# B&R Automation Studio project NAINV104C00R8L515F00 (part 17)

#### InputRef_Link.var - Change By Project
```iecst
(*2020-09-22*)
(**)
(*User Folder*)
VAR
	p_eUsrFolderStat : REFERENCE TO eUsrFolderAction;
	p_eUsrFolderStatus : REFERENCE TO eFBStatus;
END_VAR
(**)
(*Hardware Info*)
VAR
	p_eHWInfoStat : REFERENCE TO eHWInfoAction;
	p_eHWInfoStatus : REFERENCE TO eFBStatus;
	p_sHWInfoIPAddr : REFERENCE TO STRING[15];
	p_sHWInfoSubnetMask : REFERENCE TO STRING[15];
	p_udiHWInfoEthMode : REFERENCE TO UDINT;
END_VAR
(**)
(*Library Version*)
VAR
	p_eLibVerStat : REFERENCE TO eLibVerAction;
	p_eLibVerStatus : REFERENCE TO eFBStatus;
END_VAR
(**)
(*Nutek Parameter*)
VAR
	p_eNtParamStat : REFERENCE TO eNtParamAction;
	p_eNtParamStatus : REFERENCE TO eFBStatus;
END_VAR
(**)
(*Machine Parameter*)
VAR
	p_eMcParamStat : REFERENCE TO eMcParamAction;
	p_eMcParamStatus : REFERENCE TO eFBStatus;
END_VAR
(**)
(*Product Recipe*)
VAR
	p_eProdRcpStat : REFERENCE TO eProdRcpAction;
	p_eProdRcpStatus : REFERENCE TO eFBStatus;
END_VAR
(**)
(*Mp Product Recipe*)
VAR
	p_eMpProdRcpStat : REFERENCE TO eMpProdRcpAction;
	p_eMpProdRcpStatus : REFERENCE TO eFBStatus;
END_VAR
(**)
(*User Management*)
VAR
	p_eUsrMgmtStat : REFERENCE TO eUsrMgmtAction;
	p_eUsrMgmtStatus : REFERENCE TO eFBStatus;
END_VAR
(**)
(*Alarm Log*)
VAR
	p_eAlarmStat : REFERENCE TO eAlarmAction;
	p_eAlarmStatus : REFERENCE TO eFBStatus;
END_VAR
(**)
(*Hermes*)
VAR
	p_eHermesStat : REFERENCE TO eHermesAction;
	p_eHermesStatus : REFERENCE TO eFBStatus;
END_VAR
(**)
VAR
	p_eRmtHermesStat : REFERENCE TO eHermesAction;
	p_eRmtHermesStatus : REFERENCE TO eFBStatus;
END_VAR
(**)
VAR
	p_eUSHermesStat : REFERENCE TO eHermesAction;
	p_eUSHermesStatus : REFERENCE TO eFBStatus;
END_VAR
(**)
VAR
	p_eDSHermesStat : REFERENCE TO eHermesAction;
	p_eDSHermesStatus : REFERENCE TO eFBStatus;
END_VAR
(**)
(*Auto Width*)
VAR
	p_eAWStat : REFERENCE TO eAWAction;
	p_eAWStatus : REFERENCE TO eFBStatus;
END_VAR
(**)
(*User Interface*)
VAR
	p_eUIStat : REFERENCE TO eUIAction;
	p_eUIStatus : REFERENCE TO eFBStatus;
END_VAR
```

#### Act_Link.st - Change By Project
```iecst
(** 2018-12-12 **)
ACTION Act_Link:

END_ACTION
```

#### Cyclic.st - Do Not Change!!!
```iecst
(** 2019-03-29 **)
PROGRAM _CYCLIC

	IF bInitDone = FALSE THEN
		bInitDone	:= TRUE;

		Act_InitLocal;
		Act_InitGlobal;

	ELSIF bInitialDone = FALSE THEN
		bInitialDone	:= TRUE;

		Act_Initial;

	ELSE

		Act_LinkAction;
		Act_Action;
		Act_Link;
		Act_Main;

	END_IF

END_PROGRAM
```

#### Act_InitLocal.st - Do Not Change!!!
```iecst
(** 2020-09-22 **)
ACTION Act_InitLocal:

	//Input Reference Link To Local Variable
	p_eAct ACCESS ADR(eAct);
	p_tyNtParamCurr ACCESS ADR(tyNtParamCurr);
	p_tyMcParamCurr ACCESS ADR(tyMcParamCurr);

	p_bUIMismatchOverWriteConfig ACCESS ADR(bMismatchOverWriteConfig);
	p_bUITempAddrFillDone ACCESS ADR(bTempAddrFillDone);
	p_bUIChgConfigDone ACCESS ADR(bChgConfigDone);
	p_bUIOverwriteIP ACCESS ADR(bOverwriteIP);
	p_bUIOverwriteSubnet ACCESS ADR(bOverwriteSubnet);
	p_bUIOverwriteEthMode ACCESS ADR(bOverwriteEthMode);

END_ACTION
```

#### Act_Initial.st - Do Not Change!!!
```iecst
(** 2019-02-20 **)
ACTION Act_Initial:

	//Initial
	sStatTxt	:= a_sStatText[eStat];

END_ACTION
```

#### Act_Action.st - Do Not Change!!!
```iecst
(** 2019-03-25 **)
ACTION Act_Action:

	//Reset Done
	IF eStatus = Done AND p_eAct = StartupActIdle THEN
		eStat	:= StartupActIdle;
	END_IF

	//Set p_eAct
	IF eStatus = Idle THEN
		eStat	:= p_eAct;
	END_IF

END_ACTION
```

#### Act_Main.st - Change By Project
```iecst
(** 2019-03-28 **)
ACTION Act_Main:

	//Main
	CASE eStat OF

		StartupActIdle:
			IF eStatus <> Idle THEN	//Reset Data
				//Private
				eStartupStep1	:= StartupStepUsrFolder;
				bRun			:= FALSE;
				usiStep			:= 0;

				sStatTxt	:= a_sStatText[eStat];

			END_IF

			eStatus	:= Idle;

		StartupActRun:
			IF eStatus = Idle OR eStatus = Busy THEN

				eStatus	:= Busy;

				sStatTxt	:= a_sStatText[eStat];

				bRun	:= TRUE;

				CASE eStartupStep1 OF

					StartupStepUsrFolder:
						Act_Main_UsrFolder;

					StartupStepParameter:
						Act_Main_Parameter;

					StartupStepGetHWInfo:
						Act_Main_GetHWInfo;

					StartupStepLibVer:
						Act_Main_LibVer;

					StartupStepRecipe:
						Act_Main_Recipe;

					StartupStepUsrMgmt:
						Act_Main_UsrMgmt;

					StartupStepBffr:
						Act_Main_Bffr;

					StartupStepAlarm:
						Act_Main_Alarm;

					StartupStepHermes:
						Act_Main_Hermes;

					StartupStepSDOWrite:
						Act_Main_SDOWrite;

					StartupStepSetupUI:
						Act_Main_SetupUI;

					StartupStepDone:
						Act_Main_Done;

				END_CASE

				sStepTxt	:= a_sStepText[eStartupStep1];

			END_IF

	END_CASE

END_ACTION
```

#### Package Logical/Startup/Startup/Act_Main - Change By Project

#### Act_Main_UsrFolder.st
```iecst
(** 2019-05-09 **)
ACTION Act_Main_UsrFolder:

	CASE usiStep OF
		0:
			eUsrFolderAct	:= UsrFolderActCreateUsrDir;

			IF (p_eUsrFolderStatus = Done) AND (p_eUsrFolderStat = UsrFolderActCreateUsrDir) THEN

				eUsrFolderAct	:= UsrFolderActIdle;
				usiStep			:= 1;

			ELSIF p_eUsrFolderStatus = Error THEN

				eUsrFolderAct	:= UsrFolderActIdle;
				eStartupStep1	:= StartupStepParameter;

			END_IF

		1:
			eUsrFolderAct	:= UsrFolderActCreatePrivateDir;

			IF (p_eUsrFolderStatus = Done) AND (p_eUsrFolderStat = UsrFolderActCreatePrivateDir) THEN

				eUsrFolderAct	:= UsrFolderActIdle;
				usiStep			:= 2;

			ELSIF p_eUsrFolderStatus = Error THEN

				eUsrFolderAct	:= UsrFolderActIdle;
				usiStep			:= 0;
				eStartupStep1	:= StartupStepParameter;

			END_IF

		2:
			eUsrFolderAct	:= UsrFolderActCreateLogDir;

			IF (p_eUsrFolderStatus = Done) AND (p_eUsrFolderStat = UsrFolderActCreateLogDir) THEN

				eUsrFolderAct	:= UsrFolderActIdle;
				usiStep			:= 3;

			ELSIF p_eUsrFolderStatus = Error THEN

				eUsrFolderAct	:= UsrFolderActIdle;
				usiStep			:= 0;
				eStartupStep1	:= StartupStepParameter;

			END_IF

		3:
			eUsrFolderAct	:= UsrFolderActCreateLCSDir;

			IF (p_eUsrFolderStatus = Done) AND (p_eUsrFolderStat = UsrFolderActCreateLCSDir) THEN

				eUsrFolderAct	:= UsrFolderActIdle;
				usiStep			:= 0;
				eStartupStep1	:= StartupStepParameter;

			ELSIF p_eUsrFolderStatus = Error THEN

				eUsrFolderAct	:= UsrFolderActIdle;
				usiStep			:= 0;
				eStartupStep1	:= StartupStepParameter;

			END_IF

	END_CASE

END_ACTION
```

#### Act_Main_GetHWInfo.st
```iecst
(** 2020-10-05 **)
ACTION Act_Main_GetHWInfo:

	CASE usiStep OF
		0:
			eHWInfoAct	:= HWInfoActGetIPAddr;

			IF (p_eHWInfoStatus = Done) AND (p_eHWInfoStat = HWInfoActGetIPAddr) THEN

				eHWInfoAct		:= HWInfoActIdle;
				usiStep			:= 1;

			ELSIF p_eHWInfoStatus = Error THEN

				eHWInfoAct		:= HWInfoActIdle;
				eStartupStep1	:= StartupStepLibVer;

			END_IF

		1:
			eHWInfoAct	:= HWInfoActGetMacAddr;

			IF (p_eHWInfoStatus = Done) AND (p_eHWInfoStat = HWInfoActGetMacAddr) THEN

				eHWInfoAct		:= HWInfoActIdle;
				usiStep			:= 2;

			ELSIF p_eHWInfoStatus = Error THEN

				eHWInfoAct		:= HWInfoActIdle;
				usiStep			:= 0;
				eStartupStep1	:= StartupStepLibVer;

			END_IF

		2:
			eHWInfoAct	:= HWInfoActGetSubnetMask;

			IF (p_eHWInfoStatus = Done) AND (p_eHWInfoStat = HWInfoActGetSubnetMask) THEN

				eHWInfoAct		:= HWInfoActIdle;

				IF DiagCpuIsSimulated() = TRUE THEN
					usiStep			:= 0;
					eStartupStep1	:= StartupStepLibVer;
				ELSE
					usiStep			:= 3;
				END_IF

			ELSIF p_eHWInfoStatus = Error THEN

				eHWInfoAct		:= HWInfoActIdle;
				usiStep			:= 0;
				eStartupStep1	:= StartupStepLibVer;

			END_IF

		3:
			eHWInfoAct	:= HWInfoActGetEthConfigMode;

			IF (p_eHWInfoStatus = Done) AND (p_eHWInfoStat = HWInfoActGetEthConfigMode) THEN

				eHWInfoAct		:= HWInfoActIdle;

				bGetConfigDone	:= TRUE;

				IF (p_tyMcParamCurr.eNetworkMod = UDINT_TO_DINT(p_udiHWInfoEthMode))  THEN
					IF p_udiHWInfoEthMode = DINT_TO_UDINT(IPFromDHCPServer) THEN
						usiStep			:= 0;
						eStartupStep1	:= StartupStepLibVer;
					ELSE
						IF (p_tyMcParamCurr.sIPAddr <> p_sHWInfoIPAddr) OR (p_tyMcParamCurr.sSubnetMask <> p_sHWInfoSubnetMask) THEN
							IF p_bUITempAddrFillDone AND p_bUIMismatchOverWriteConfig THEN
								IF (p_tyMcParamCurr.sIPAddr <> p_sHWInfoIPAddr) THEN
									usiStep			:= 5;  //mismatch ip
								ELSE
									usiStep			:= 6;  //mismatch subnet
								END_IF
							END_IF
						ELSE
							usiStep			:= 0;
							eStartupStep1	:= StartupStepLibVer;
						END_IF
					END_IF

				ELSE
					IF p_bUITempAddrFillDone AND p_bUIMismatchOverWriteConfig THEN
						usiStep			:= 4;
					END_IF
				END_IF

			ELSIF p_eHWInfoStatus = Error THEN

				eHWInfoAct		:= HWInfoActIdle;
				usiStep			:= 0;
				eStartupStep1	:= StartupStepLibVer;

			END_IF

		4:
			eHWInfoAct	:= HWInfoActSetEthConfigMode;

			IF (p_eHWInfoStatus = Done) AND (p_eHWInfoStat = HWInfoActSetEthConfigMode) THEN

				eHWInfoAct		:= HWInfoActIdle;

				IF (p_tyMcParamCurr.eNetworkMod = IPFromDHCPServer) THEN
					usiStep			:= 7;
					bMismatchSetConfigDone	:= TRUE;
				ELSE
					usiStep			:= 5;
				END_IF

			ELSIF p_eHWInfoStatus = Error THEN

				eHWInfoAct		:= HWInfoActIdle;
				usiStep			:= 0;
				eStartupStep1	:= StartupStepLibVer;

			END_IF

		5:
			eHWInfoAct	:= HWInfoActSetIPAddr;

			IF (p_eHWInfoStatus = Done) AND (p_eHWInfoStat = HWInfoActSetIPAddr) THEN

				eHWInfoAct		:= HWInfoActIdle;

				IF (p_tyMcParamCurr.sSubnetMask <> p_sHWInfoSubnetMask) THEN
					usiStep			:= 6;
				ELSE
					usiStep			:= 7;
					bMismatchSetConfigDone	:= TRUE;
				END_IF

			ELSIF p_eHWInfoStatus = Error THEN

				eHWInfoAct		:= HWInfoActIdle;
				usiStep			:= 0;
				eStartupStep1	:= StartupStepLibVer;

			END_IF

		6:
			eHWInfoAct	:= HWInfoActSetSubnetMask;

			IF (p_eHWInfoStatus = Done) AND (p_eHWInfoStat = HWInfoActSetSubnetMask) THEN

				eHWInfoAct		:= HWInfoActIdle;
				usiStep			:= 7;

				bMismatchSetConfigDone	:= TRUE;

			ELSIF p_eHWInfoStatus = Error THEN

				eHWInfoAct		:= HWInfoActIdle;
				usiStep			:= 0;
				eStartupStep1	:= StartupStepLibVer;

			END_IF

		7:
			IF p_bUIChgConfigDone THEN
				IF p_bUIOverwriteEthMode THEN
					usiStep			:= 8; //Overwrite Network Mode
				ELSIF p_bUIOverwriteIP THEN
					usiStep			:= 9; //Overwrite IP
				ELSIF p_bUIOverwriteSubnet THEN
					usiStep			:= 10; //Overwrite Subnet
				ELSE
					usiStep			:= 12; //Load Machine Setting
				END_IF
			END_IF

		8:
			eHWInfoAct	:= HWInfoActSetEthConfigMode;

			IF (p_eHWInfoStatus = Done) AND (p_eHWInfoStat = HWInfoActSetEthConfigMode) THEN

				eHWInfoAct		:= HWInfoActIdle;

				IF p_bUIOverwriteIP THEN
					usiStep			:= 9;
				ELSIF p_bUIOverwriteSubnet THEN
					usiStep			:= 10;
				ELSE
					usiStep			:= 11;
				END_IF

			ELSIF p_eHWInfoStatus = Error THEN

				eHWInfoAct		:= HWInfoActIdle;
				usiStep			:= 0;
				eStartupStep1	:= StartupStepLibVer;

			END_IF

		9:
			eHWInfoAct	:= HWInfoActSetIPAddr;

			IF (p_eHWInfoStatus = Done) AND (p_eHWInfoStat = HWInfoActSetIPAddr) THEN

				eHWInfoAct		:= HWInfoActIdle;

				IF p_bUIOverwriteSubnet THEN
					usiStep			:= 10;
				ELSE
					usiStep			:= 11;
				END_IF

			ELSIF p_eHWInfoStatus = Error THEN

				eHWInfoAct		:= HWInfoActIdle;
				usiStep			:= 0;
				eStartupStep1	:= StartupStepLibVer;

			END_IF

		10:
			eHWInfoAct	:= HWInfoActSetSubnetMask;

			IF (p_eHWInfoStatus = Done) AND (p_eHWInfoStat = HWInfoActSetSubnetMask) THEN

				eHWInfoAct		:= HWInfoActIdle;
				usiStep			:= 11;

			ELSIF p_eHWInfoStatus = Error THEN

				eHWInfoAct		:= HWInfoActIdle;
				usiStep			:= 0;
				eStartupStep1	:= StartupStepLibVer;

			END_IF

		11:

			eMcParamAct	:= McParamActWrite;

			IF (p_eMcParamStatus = Done) AND (p_eMcParamStat = McParamActWrite) THEN

				eMcParamAct		:= McParamActIdle;

				usiStep			:= 12;

			ELSIF p_eMcParamStatus = Error THEN

				eMcParamAct		:= McParamActIdle;
				usiStep			:= 0;
				eStartupStep1	:= StartupStepLibVer;

			END_IF

		12:
			eHWInfoAct	:= HWInfoActGetIPAddr;

			IF (p_eHWInfoStatus = Done) AND (p_eHWInfoStat = HWInfoActGetIPAddr) THEN

				eHWInfoAct		:= HWInfoActIdle;
				usiStep			:= 13;

			ELSIF p_eHWInfoStatus = Error THEN

				eHWInfoAct		:= HWInfoActIdle;
				usiStep			:= 0;
				eStartupStep1	:= StartupStepLibVer;

			END_IF

		13:
			eHWInfoAct	:= HWInfoActGetSubnetMask;

			IF (p_eHWInfoStatus = Done) AND (p_eHWInfoStat = HWInfoActGetSubnetMask) THEN

				eHWInfoAct		:= HWInfoActIdle;
				usiStep			:= 0;
				eStartupStep1	:= StartupStepLibVer;

			ELSIF p_eHWInfoStatus = Error THEN

				eHWInfoAct		:= HWInfoActIdle;
				usiStep			:= 0;
				eStartupStep1	:= StartupStepLibVer;

			END_IF

	END_CASE

END_ACTION
```

#### Act_Main_LibVer.st
```iecst
(** 2019-03-28 **)
ACTION Act_Main_LibVer:

	CASE usiStep OF
		0:
			eLibVerAct	:= LibVerActCreateDir;

			IF (p_eLibVerStatus = Done) AND (p_eLibVerStat = LibVerActCreateDir) THEN

				eLibVerAct		:= LibVerActIdle;
				usiStep			:= 1;

			ELSIF p_eLibVerStatus = Error THEN

				eLibVerAct		:= LibVerActIdle;
				eStartupStep1	:= StartupStepRecipe;

			END_IF

		1:
			eLibVerAct	:= LibVerActReadChk;

			IF (p_eLibVerStatus = Done) AND (p_eLibVerStat = LibVerActReadChk) THEN

				eLibVerAct		:= LibVerActIdle;
				usiStep			:= 0;
				eStartupStep1	:= StartupStepRecipe;

			ELSIF p_eLibVerStatus = Error THEN

				eLibVerAct		:= LibVerActIdle;
				usiStep			:= 0;
				eStartupStep1	:= StartupStepRecipe;

			END_IF

	END_CASE

END_ACTION
```

#### Act_Main_Parameter.st
```iecst
(** 2019-03-28 **)
ACTION Act_Main_Parameter:

	CASE usiStep OF
		0:
			eNtParamAct	:= NtParamActCreateDir;

			IF (p_eNtParamStatus = Done) AND (p_eNtParamStat = NtParamActCreateDir) THEN

				eNtParamAct			:= NtParamActIdle;
				usiStep				:= 1;

			ELSIF p_eNtParamStatus = Error THEN

				bNtSettingsLoadDone	:= TRUE;
				eNtParamAct			:= NtParamActIdle;
				usiStep				:= 2;

			END_IF

		1:
			eNtParamAct	:= NtParamActRead;

			IF (p_eNtParamStatus = Done) AND (p_eNtParamStat = NtParamActRead) THEN

				bNtSettingsLoadDone	:= TRUE;
				eNtParamAct			:= NtParamActIdle;
				usiStep				:= 2;

			ELSIF p_eNtParamStatus = Error THEN

				bNtSettingsLoadDone	:= TRUE;
				eNtParamAct			:= NtParamActIdle;
				usiStep				:= 2;

			END_IF

		2:
			eMcParamAct	:= McParamActCreateDir;

			IF (p_eMcParamStatus = Done) AND (p_eMcParamStat = McParamActCreateDir) THEN

				eMcParamAct		:= McParamActIdle;
				usiStep			:= 3;

			ELSIF p_eMcParamStatus = Error THEN

				eMcParamAct		:= McParamActIdle;
				usiStep			:= 0;
				eStartupStep1	:= StartupStepGetHWInfo;

			END_IF

		3:
			eMcParamAct	:= McParamActRead;

			IF (p_eMcParamStatus = Done) AND (p_eMcParamStat = McParamActRead) THEN

				eMcParamAct		:= McParamActIdle;
				usiStep			:= 0;
				eStartupStep1	:= StartupStepGetHWInfo;

			ELSIF p_eMcParamStatus = Error THEN

				eMcParamAct		:= McParamActIdle;
				usiStep			:= 0;
				eStartupStep1	:= StartupStepGetHWInfo;

			END_IF

	END_CASE

END_ACTION
```

#### Act_Main_Recipe.st
```iecst
(** 2019-05-04 **)
ACTION Act_Main_Recipe:

	CASE usiStep OF
		0:
			eProdRcpAct	:= ProdRcpActCreateDir;

			IF (p_eProdRcpStatus = Done) AND (p_eProdRcpStat = ProdRcpActCreateDir) THEN

				eProdRcpAct		:= ProdRcpActIdle;
				usiStep			:= 1;

			ELSIF p_eProdRcpStatus = Error THEN

				eProdRcpAct		:= ProdRcpActIdle;
				usiStep			:= 10;

			END_IF

		1:
			eProdRcpAct	:= ProdRcpActGetList;

			IF (p_eProdRcpStatus = Done) AND (p_eProdRcpStat = ProdRcpActGetList) THEN

				eProdRcpAct		:= ProdRcpActIdle;
				usiStep			:= 2;

			ELSIF p_eProdRcpStatus = Error THEN

				eProdRcpAct		:= ProdRcpActIdle;
				usiStep			:= 10;

			END_IF

		2:
			eProdRcpAct	:= ProdRcpActReadCurrRcp;

			IF (p_eProdRcpStatus = Done) AND (p_eProdRcpStat = ProdRcpActReadCurrRcp) THEN

				eProdRcpAct		:= ProdRcpActIdle;
				usiStep			:= 10;

			ELSIF p_eProdRcpStatus = Error THEN

				eProdRcpAct		:= ProdRcpActIdle;
				usiStep			:= 10;

			END_IF

		10:
			eMpProdRcpAct	:= MpProdRcpActCreateDir;

			IF (p_eMpProdRcpStatus = Done) AND (p_eMpProdRcpStat = MpProdRcpActCreateDir) THEN

				eMpProdRcpAct	:= MpProdRcpActIdle;
				usiStep			:= 0;
				eStartupStep1	:= StartupStepUsrMgmt;

			ELSIF p_eProdRcpStatus = Error THEN

				eMpProdRcpAct	:= MpProdRcpActIdle;
				usiStep			:= 0;
				eStartupStep1	:= StartupStepUsrMgmt;

			END_IF

	END_CASE

END_ACTION
```

#### Act_Main_UsrMgmt.st
```iecst
(** 2019-03-28 **)
ACTION Act_Main_UsrMgmt:

	CASE usiStep OF
		0:
			eUsrMgmtAct	:= UsrMgmtActCreateDir;

			IF (p_eUsrMgmtStatus = Done) AND (p_eUsrMgmtStat = UsrMgmtActCreateDir) THEN

				eUsrMgmtAct		:= UsrMgmtActIdle;
				usiStep			:= 1;

			ELSIF p_eUsrMgmtStatus = Error THEN

				eUsrMgmtAct		:= UsrMgmtActIdle;
				eStartupStep1	:= StartupStepBffr;

			END_IF

		1:
			eUsrMgmtAct	:= UsrMgmtActReadData;

			IF (p_eUsrMgmtStatus = Done) AND (p_eUsrMgmtStat = UsrMgmtActReadData) THEN

				eUsrMgmtAct		:= UsrMgmtActIdle;
				usiStep			:= 2;

			ELSIF p_eUsrMgmtStatus = Error THEN

				eUsrMgmtAct		:= UsrMgmtActIdle;
				usiStep			:= 0;
				eStartupStep1	:= StartupStepBffr;

			END_IF

		2:
			eUsrMgmtAct	:= UsrMgmtActLogout;

			IF (p_eUsrMgmtStatus = Done) AND (p_eUsrMgmtStat = UsrMgmtActLogout) THEN

				eUsrMgmtAct		:= UsrMgmtActIdle;
				usiStep			:= 0;
				eStartupStep1	:= StartupStepBffr;

			ELSIF p_eUsrMgmtStatus = Error THEN

				eUsrMgmtAct		:= UsrMgmtActIdle;
				usiStep			:= 0;
				eStartupStep1	:= StartupStepBffr;

			END_IF

	END_CASE

END_ACTION
```

#### Act_Main_Bffr.st
```iecst
(** 2013-04-26 **)
ACTION Act_Main_Bffr:

	eStartupStep1	:= StartupStepAlarm;

END_ACTION
```

#### Act_Main_Alarm.st
```iecst
(** 2019-03-28 **)
ACTION Act_Main_Alarm:

	CASE usiStep OF
		0:
			eAlarmAct	:= AlarmActCreateDir;

			IF (p_eAlarmStatus = Done) AND (p_eAlarmStat = AlarmActCreateDir) THEN

				eAlarmAct		:= AlarmActIdle;
				usiStep			:= 1;

			ELSIF p_eAlarmStatus = Error THEN

				eAlarmAct		:= AlarmActIdle;
				usiStep			:= 0;
				eStartupStep1	:= StartupStepHermes;

			END_IF

		1:
			eAlarmAct	:= AlarmActDeleteOldLog;

			IF (p_eAlarmStatus = Done) AND (p_eAlarmStat = AlarmActDeleteOldLog) THEN

				eAlarmAct		:= AlarmActIdle;
				usiStep			:= 2;

			ELSIF p_eAlarmStatus = Error THEN

				eAlarmAct		:= AlarmActIdle;
				usiStep			:= 0;
				eStartupStep1	:= StartupStepHermes;

			END_IF

		2:
			eAlarmAct	:= AlarmActReadHistory;

			IF (p_eAlarmStatus = Done) AND (p_eAlarmStat = AlarmActReadHistory) THEN

				eAlarmAct		:= AlarmActIdle;
				usiStep			:= 3;

			ELSIF p_eAlarmStatus = Error THEN

				eAlarmAct		:= AlarmActIdle;
				usiStep			:= 0;
				eStartupStep1	:= StartupStepHermes;

			END_IF

		3:
			eAlarmAct	:= AlarmActBGStartLog;

			IF (p_eAlarmStatus = Done) AND (p_eAlarmStat = AlarmActBGStartLog) THEN

				eAlarmAct		:= AlarmActIdle;
				usiStep			:= 0;
				eStartupStep1	:= StartupStepHermes;

			ELSIF p_eAlarmStatus = Error THEN

				eAlarmAct		:= AlarmActIdle;
				usiStep			:= 0;
				eStartupStep1	:= StartupStepHermes;

			END_IF

	END_CASE

END_ACTION
```

#### Act_Main_Hermes.st
```iecst
(** 2019-05-04 **)
ACTION Act_Main_Hermes:

	CASE usiStep OF
		0:
			eHermesAct	:= HermesActCreateDir;

			IF (p_eHermesStatus = Done) AND (p_eHermesStat = HermesActCreateDir) THEN

				eHermesAct		:= HermesActIdle;
				usiStep			:= 1;

			ELSIF p_eHermesStatus = Error THEN

				eHermesAct		:= HermesActIdle;
				usiStep			:= 10;

			END_IF

		1:
			eHermesAct	:= HermesActReadRetainLane1; //HermesActReadRetain;

			IF (p_eHermesStatus = Done) AND (p_eHermesStat = HermesActReadRetainLane1) THEN

				eHermesAct		:= HermesActIdle;
				usiStep			:= 2;

			ELSIF p_eHermesStatus = Error THEN

				eHermesAct		:= HermesActIdle;
				usiStep			:= 10;

			END_IF

		2:
			eHermesAct	:= HermesActReadConfig;

			IF (p_eHermesStatus = Done) AND (p_eHermesStat = HermesActReadConfig) THEN

				eHermesAct		:= HermesActIdle;
				usiStep			:= 10;

			ELSIF p_eHermesStatus = Error THEN

				eHermesAct		:= HermesActIdle;
				usiStep			:= 10;

			END_IF

		10:
			eRmtHermesAct	:= HermesActDeleteOldLog;

			IF (p_eRmtHermesStatus = Done) AND (p_eRmtHermesStat = HermesActDeleteOldLog) THEN

				eRmtHermesAct	:= HermesActIdle;
				usiStep			:= 20;

			ELSIF p_eRmtHermesStatus = Error THEN

				eRmtHermesAct	:= HermesActIdle;
				usiStep			:= 20;

			END_IF
		20:
			eDSHermesAct	:= HermesActReadRetain;

			IF (p_eDSHermesStatus = Done) AND (p_eDSHermesStat = HermesActReadRetain) THEN

				eDSHermesAct	:= HermesActIdle;
				usiStep			:= 21;

			ELSIF p_eDSHermesStatus = Error THEN //when there is no Retain file created, then p_eDSHermesStatus will be error, skip to startup)

				eDSHermesAct	:= HermesActIdle;
				usiStep			:= 21;

			END_IF

		21:
			eDSHermesAct	:= HermesActDeleteOldLog;

			IF (p_eDSHermesStatus = Done) AND (p_eDSHermesStat = HermesActDeleteOldLog) THEN

				eDSHermesAct	:= HermesActIdle;
				usiStep			:= 30;

			ELSIF p_eDSHermesStatus = Error THEN

				eDSHermesAct	:= HermesActIdle;
				usiStep			:= 30;

			END_IF

		30:
			eRmtHermesAct	:= HermesActDeleteOldLog;

			IF (p_eRmtHermesStatus = Done) AND (p_eRmtHermesStat = HermesActDeleteOldLog) THEN

				eRmtHermesAct	:= HermesActIdle;
				usiStep			:= 0;
				eStartupStep1	:= StartupStepSetupUI;
			ELSIF p_eRmtHermesStatus = Error THEN

				eRmtHermesAct	:= HermesActIdle;
				usiStep			:= 0;
				eStartupStep1	:= StartupStepSetupUI;
			END_IF

//		40:
//			eSvyHermesAct	:= HermesActDeleteOldLog;
//
//			IF (p_eSvyHermesStatus = Done) AND (p_eSvyHermesStat = HermesActDeleteOldLog) THEN
//
//				eSvyHermesAct	:= HermesActIdle;
//				usiStep			:= 41;
//
//			ELSIF p_eSvyHermesStatus = Error THEN
//
//				eSvyHermesAct	:= HermesActIdle;
//				usiStep			:= 41;
//
//			END_IF

//		41:
//			bWaitDecision := TRUE;
//
//			IF p_bUIReadWorkOrder THEN
//				eSvyHermesAct	:= HermesActReadRetain;
//
//				IF (p_eSvyHermesStatus = Done) AND (p_eSvyHermesStat = HermesActReadRetain) THEN
//
//					eSvyHermesAct	:= HermesActIdle;
//					usiStep			:= 0;
//					eStartupStep1	:= StartupStepSetupUI;
//					bWaitDecision := FALSE;
//
//				ELSIF p_eSvyHermesStatus = Error THEN
//
//					eSvyHermesAct	:= HermesActIdle;
//					usiStep			:= 0;
//					eStartupStep1	:= StartupStepSetupUI;
//					bWaitDecision := FALSE;
//
//				END_IF
//
//			ELSIF p_bUISkipWorkOrder THEN
//				usiStep			:= 0;
//				eStartupStep1	:= StartupStepSetupUI;
//				bWaitDecision := FALSE;
//			END_IF
	END_CASE

END_ACTION
```

#### Act_Main_SDOWrite.st
```iecst
(** 2019-10-21 **)
ACTION Act_Main_SDOWrite:

	CASE usiStep OF
		0:
//			eAWAct	:= AWActBGStartModOKChk;
//
//			IF (p_eAWStatus = Done) AND (p_eAWStat = AWActBGStartModOKChk) THEN
//
//				eAWAct		:= AWActIdle;
//				usiStep		:= 0;
//				eStartupStep1 := StartupStepSetupUI;
//
//			ELSIF p_eAWStatus = Error THEN
//
//				eAWAct		:= AWActIdle;
//				usiStep		:= 0;
				eStartupStep1 := StartupStepSetupUI;

//			END_IF

	END_CASE

END_ACTION
```

#### Act_Main_SetupUI.st
```iecst
(** 2019-03-28 **)
ACTION Act_Main_SetupUI:

	CASE usiStep OF
		0:
			eUIAct	:= UIActInitial;

			IF (p_eUIStatus = Done) AND (p_eUIStat = UIActInitial) THEN

				eUIAct			:= UIActIdle;
				eStartupStep1	:= StartupStepDone;
				bUISettingsLoadDone := TRUE;
			ELSIF p_eUIStatus = Error THEN

				eUIAct			:= UIActIdle;
				eStartupStep1	:= StartupStepDone;
				bUISettingsLoadDone := TRUE;
			END_IF

	END_CASE

END_ACTION
```

#### Act_Main_Done.st
```iecst
(** 2018-12-26 **)
ACTION Act_Main_Done:

	eStatus	:= Done;

END_ACTION
```

#### InputRef.var - Do Not Change!!!
```iecst
(*2020-09-22*)
(**)
(*General*)
VAR
	p_eAct : REFERENCE TO eStartupAction;
	p_tyNtParamCurr : REFERENCE TO tyNtParam;
	p_tyMcParamCurr : REFERENCE TO tyMcParam;
	p_bUIMismatchOverWriteConfig : REFERENCE TO BOOL;
	p_bUITempAddrFillDone : REFERENCE TO BOOL;
	p_bUIChgConfigDone : REFERENCE TO BOOL;
	p_bUIOverwriteIP : REFERENCE TO BOOL;
	p_bUIOverwriteSubnet : REFERENCE TO BOOL;
	p_bUIOverwriteEthMode : REFERENCE TO BOOL;
END_VAR
```

#### Local.var - Do Not Change!!!
```iecst
(*2020-09-22*)
(**)
(*Local Action, State & Status*)
VAR
	eAct : eStartupAction := StartupActIdle;
	eStat : eStartupAction := StartupActIdle;
	eStatus : eFBStatus := Idle;
	sStatTxt : STRING[200] := '';
	a_sStatText : ARRAY[0..50] OF STRING[200] := ['Idling','Running Startup',49('')];
END_VAR
(**)
(*Local Alarm*)
(**)
(*Local Output*)
VAR
	bRun : BOOL;
	eUsrFolderAct : eUsrFolderAction;
	eHWInfoAct : eHWInfoAction;
	eLibVerAct : eLibVerAction;
	eNtParamAct : eNtParamAction;
	eMcParamAct : eMcParamAction;
	eProdRcpAct : eProdRcpAction;
	eMpProdRcpAct : eMpProdRcpAction;
	eUsrMgmtAct : eUsrMgmtAction;
	eAlarmAct : eAlarmAction;
	eUIAct : eUIAction;
	eAWAct : eAWAction;
	eHermesAct : eHermesAction;
	eRmtHermesAct : eHermesAction;
	eUSHermesAct : eHermesAction;
	eDSHermesAct : eHermesAction;
	eStartupStep1 : eStartupStep;
	bNtSettingsLoadDone : BOOL := FALSE;
	bUISettingsLoadDone : BOOL;
	sStepTxt : STRING[80];
	a_sStepText : ARRAY[0..11] OF STRING[80] := ['Creating User Folder','Reading Parameter','Getting Hardware Info','Checking Library Version','Reading Recipe List','Reading User Management List','Reading Buffer / Magazine Data','Setting Up Alarm','Setting Up Hermes','Writing Data To Servo Motor','Setting Up User Interface','Done'];
END_VAR
(**)
(*Local Input*)
VAR
	bMismatchOverWriteConfig : BOOL;
	bTempAddrFillDone : BOOL;
	bChgConfigDone : BOOL;
	bOverwriteIP : BOOL;
	bOverwriteSubnet : BOOL;
	bOverwriteEthMode : BOOL;
	bGetConfigDone : BOOL;
	bMismatchSetConfigDone : BOOL;
	tyNtParamCurr : tyNtParam;
	tyMcParamCurr : tyMcParam;
END_VAR
(**)
(*Local*)
VAR
	bInitDone : BOOL;
	bInitialDone : BOOL;
	usiStep : USINT;
END_VAR
```

### General.typ - Do Not Change!!!
```iecst
(*2018-12-07*)
(**)
(*Action*)

TYPE
	eGeneralAction :
		(
		GeneralActIdle,
		GeneralActIPValid
		);
END_TYPE
```

### General.var - Change By Project
```iecst
(*2019-03-25*)
(**)
(*Action & State & Status*)
VAR
	p_GeneralStat : UDINT;
	p_GeneralStatus : UDINT;
	p_GeneralStatTxt : UDINT;
END_VAR
(**)
(*Alarm*)
(**)
(*Output*)
VAR
	p_GeneralIPPart : UDINT;
	p_GeneralIPValid : UDINT;
END_VAR
```

### Program Logical/General/General (IEC) - 1.00.0 - 

#### InputRef.var
```iecst
(*2019-03-25*)
(**)
(*Configuration*)
VAR
	p_eAct : REFERENCE TO eGeneralAction;
	p_sIPAddr : REFERENCE TO STRING[15];
	p_bNtSettingsLoadDone : REFERENCE TO BOOL;
END_VAR
```

#### Local.var
```iecst
(*2019-04-30*)
(**)
(*Local Action, State & Status*)
VAR
	eAct : eGeneralAction := GeneralActIdle;
	eStat : eGeneralAction := GeneralActIdle;
	eStatus : eFBStatus := Idle;
	sStatTxt : STRING[200] := '';
	a_sStatText : ARRAY[0..50] OF STRING[200] := ['Idling','Checking IP Validity',49('')];
END_VAR
(**)
(*Local Alarm*)
(**)
(*Local Output*)
VAR
	a_iIPPart : ARRAY[1..4] OF INT;
	bIPValid : BOOL;
END_VAR
(**)
(*Local Input*)
VAR
	sIPAddr : STRING[15];
	bNtSettingsLoadDone : BOOL := TRUE;
END_VAR
(**)
(*Local*)
VAR
	bInitDone : BOOL;
	bInitialDone : BOOL;
END_VAR
```

#### Act_Action.st
```iecst
(** 2019-03-25 **)
ACTION Act_Action:

	//Reset Done
	IF eStatus = Done AND p_eAct = GeneralActIdle THEN
		eStat	:= GeneralActIdle;
	END_IF

	//Set p_eAct
	IF eStatus = Idle THEN
		eStat	:= p_eAct;
	END_IF

END_ACTION
```

#### Act_InitGlobal.st
```iecst
(** 201-03-22 **)
ACTION Act_InitGlobal:

	(* Always Change If Project Change *)

	//Pass Data To Link

	//Pass Data To Internal Use
	p_bNtSettingsLoadDone ACCESS p_StartupNtSettingsLoadDone;

	(* Always Change If Project Change *)

END_ACTION
```

#### Act_InitLocal.st
```iecst
(** 2019-03-25 **)
ACTION Act_InitLocal:

	//Input Reference Link To Local Variable
	p_eAct ACCESS ADR(eAct);
	p_sIPAddr ACCESS ADR(sIPAddr);
	p_bNtSettingsLoadDone ACCESS ADR(bNtSettingsLoadDone);

END_ACTION
```

#### Act_Link.st
```iecst
(** 2018-12-07 **)
ACTION Act_Link:

END_ACTION
```

#### Act_Main.st
```iecst
(** 2019-01-02 **)
ACTION Act_Main:

	//Main
	CASE eStat OF

		GeneralActIdle:
			IF eStatus <> Idle THEN	//Reset Data
				//Private
				memset(ADR(a_iIPPart), 0, SIZEOF(a_iIPPart));
				bIPValid	:= FALSE;

				sStatTxt	:= a_sStatText[eStat];

			END_IF

			eStatus	:= Idle;

		GeneralActIPValid:
			IF eStatus = Idle OR eStatus = Busy THEN

				sStatTxt	:= a_sStatText[eStat];

				bIPValid	:= fIPValid(p_sIPAddr , ADR(a_iIPPart));

				eStatus	:= Done;

			END_IF

	END_CASE

END_ACTION
```

#### Cyclic.st
```iecst
(** 2019-03-29 **)
PROGRAM _CYCLIC

	IF bInitDone = FALSE THEN
		bInitDone	:= TRUE;

		Act_InitLocal;
		Act_InitGlobal;

	ELSIF bInitialDone = FALSE THEN
		IF p_bNtSettingsLoadDone = TRUE THEN
			bInitialDone	:= TRUE;

			Act_Initial;
		END_IF

	ELSE

		Act_LinkAction;
		Act_Action;
		Act_Link;
		Act_Main;

	END_IF

END_PROGRAM
```

#### Init.st
```iecst
(** 2019-03-25 **)
PROGRAM _INIT

	(* Always Change If Project Change *)

	//Pass Address To Global Address For External Use
	//Action, State & Status
	p_GeneralStat		:= ADR(eStat);
	p_GeneralStatus		:= ADR(eStatus);
	p_GeneralStatTxt	:= ADR(sStatTxt);

	//Alarm

	//Output
	p_GeneralIPPart		:= ADR(a_iIPPart);
	p_GeneralIPValid	:= ADR(bIPValid);

	(* Always Change If Project Change *)

END_PROGRAM
```

### UsrFolder.typ - Do Not Change!!!
```iecst
(*2019-05-09*)
(**)
(*Action*)

TYPE
	eUsrFolderAction :
		(
		UsrFolderActIdle,
		UsrFolderActCreateUsrDir,
		UsrFolderActCreatePrivateDir,
		UsrFolderActCreateLogDir,
		UsrFolderActCreateLCSDir
		);
END_TYPE
```

### UsrFolder.var - Change By Project
```iecst
(*2019-03-25*)
(**)
(*Action & State & Status*)
VAR
	p_UsrFolderStat : UDINT;
	p_UsrFolderStatus : UDINT;
	p_UsrFolderStatTxt : UDINT;
END_VAR
(**)
(*Alarm*)
VAR
	p_UsrFolderAlmData : UDINT;
END_VAR
(**)
(*Output*)
```

### Program Logical/UsrFolder/UsrFolder (IEC, version 1.00.0) - 1.00.0 - NtFileIO v5.00.0

#### Init.st - Change By Project
```iecst
(** 2019-03-25 **)
PROGRAM _INIT

	(* Always Change If Project Change *)

	//Pass Address To Global Address For External Use
	//Action, State & Status
	p_UsrFolderStat		:= ADR(eStat);
	p_UsrFolderStatus	:= ADR(eStatus);
	p_UsrFolderStatTxt	:= ADR(sStatTxt);

	//Alarm
	p_UsrFolderAlmData	:= ADR(tyAlmData);

	//Output

	(* Always Change If Project Change *)

END_PROGRAM
```

#### Act_InitGlobal.st - Change By Project
```iecst
(** 2019-03-25 **)
ACTION Act_InitGlobal:

	(* Always Change If Project Change *)

	//Pass Data To Link

	//Pass Data To Internal Use
	p_udiRstErr ACCESS p_RstErrReset;
	p_eAct ACCESS p_StartupUsrFolderAct;
	p_sProgNm ACCESS p_NtParamUsrFolderProgNm;

	(* Always Change If Project Change *)

END_ACTION
```

#### Act_LinkAction.st - Change By Project
```iecst
(** 2019-03-29 **)
ACTION Act_LinkAction:

END_ACTION
```

#### Cyclic.st - Do Not Change!!!
```iecst
(** 2019-03-29 **)
PROGRAM _CYCLIC

	IF bInitDone = FALSE THEN
		bInitDone	:= TRUE;

		Act_InitLocal;
		Act_InitGlobal;

	ELSIF bInitialDone = FALSE THEN
		bInitialDone	:= TRUE;

		Act_Initial;

	ELSE

		Act_RstErr;
		Act_LinkAction;
		Act_Action;
		Act_Link;
		Act_Main;
		Act_Alarm;

	END_IF

END_PROGRAM
```

#### Act_InitLocal.st - Do Not Change!!!
```iecst
(** 2019-03-25 **)
ACTION Act_InitLocal:

	//Input Reference Link To Local Variable
	p_eAct ACCESS ADR(eAct);
	p_udiRstErr ACCESS ADR(udiRstErr);
	p_sProgNm ACCESS ADR(sProgNm);

END_ACTION
```

#### Act_Initial.st - Do Not Change!!!
```iecst
(** 2019-05-09 **)
ACTION Act_Initial:

	//Initial
	sStatTxt	:= a_sStatText[eStat];

	fbDirCreate1.sDevice	:= 'F';
	fbDirCreate1.sDirName	:= 'User';
	fbDirCreate1(bEn := FALSE);

	fbDirCreate2.sDevice	:= 'F';
	fbDirCreate2.sDirName	:= 'Private';
	fbDirCreate2(bEn := FALSE);

	fbDirCreate3.sDevice	:= 'User';
	fbDirCreate3.sDirName	:= 'Log';
	fbDirCreate3(bEn := FALSE);

	fbDirCreate4.sDevice	:= 'User';
	fbDirCreate4.sDirName	:= 'LCS';
	fbDirCreate4(bEn := FALSE);

END_ACTION
```

#### Act_Action.st - Do Not Change!!!
```iecst
(** 2019-03-25 **)
ACTION Act_Action:

	//Reset Error
	IF (eStatus = Error) AND bRstErr THEN
		p_eAct	:= UsrFolderActIdle;
		eStat	:= UsrFolderActIdle;
	END_IF

	//Reset Done. Done Only Exist One Cycle.
	IF eStatus = Done AND p_eAct = UsrFolderActIdle THEN
		eStat	:= UsrFolderActIdle;
	END_IF

	//Set p_eAct
	IF eStatus = Idle THEN
		eStat	:= p_eAct;
	END_IF

END_ACTION
```

#### Act_Main.st - Do Not Change!!!
```iecst
(** 2019-05-09 **)
ACTION Act_Main:

	//Main
	CASE eStat OF

		UsrFolderActIdle:
			IF eStatus <> Idle THEN	//Reset Data
				//Private
				fbDirCreate1(bEn := FALSE);
				fbDirCreate2(bEn := FALSE);
				fbDirCreate3(bEn := FALSE);
				fbDirCreate4(bEn := FALSE);

				sStatTxt	:= a_sStatText[eStat];

			END_IF

			eStatus	:= Idle;

		UsrFolderActCreateUsrDir:
			IF eStatus = Idle OR eStatus = Busy THEN

				eStatus	:= Busy;

				sStatTxt	:= a_sStatText[eStat];

				fbDirCreate1(bEn := TRUE);
				IF fbDirCreate1.udiStatus = 0 THEN
					eStatus		:= Done;
				ELSIF fbDirCreate1.udiStatus < 65534 THEN
					eStatus		:= Error;

					IF fbDirCreate1.udiStatus = 1908 THEN
						udiStatus	:= 10000;	//Creating User Directory Error
					ELSE
						udiStatus	:= fbDirCreate1.udiStatus;
					END_IF
				END_IF

			END_IF

		UsrFolderActCreatePrivateDir:
			IF eStatus = Idle OR eStatus = Busy THEN

				eStatus	:= Busy;

				sStatTxt	:= a_sStatText[eStat];

				fbDirCreate2(bEn := TRUE);
				IF fbDirCreate2.udiStatus = 0 THEN
					eStatus		:= Done;
				ELSIF fbDirCreate2.udiStatus < 65534 THEN
					eStatus		:= Error;

					IF fbDirCreate2.udiStatus = 1908 THEN
						udiStatus	:= 10001;	//Creating Private Directory Error
					ELSE
						udiStatus	:= fbDirCreate2.udiStatus;
					END_IF
				END_IF

			END_IF

		UsrFolderActCreateLogDir:
			IF eStatus = Idle OR eStatus = Busy THEN

				eStatus	:= Busy;

				sStatTxt	:= a_sStatText[eStat];

				fbDirCreate3(bEn := TRUE);
				IF fbDirCreate3.udiStatus = 0 THEN
					eStatus		:= Done;
				ELSIF fbDirCreate3.udiStatus < 65534 THEN
					eStatus		:= Error;

					IF fbDirCreate3.udiStatus = 1908 THEN
						udiStatus	:= 10002;	//Creating Log Directory Error
					ELSE
						udiStatus	:= fbDirCreate3.udiStatus;
					END_IF
				END_IF

			END_IF

		UsrFolderActCreateLCSDir:
			IF eStatus = Idle OR eStatus = Busy THEN

				eStatus	:= Busy;

				sStatTxt	:= a_sStatText[eStat];

				fbDirCreate4(bEn := TRUE);
				IF fbDirCreate4.udiStatus = 0 THEN
					eStatus		:= Done;
				ELSIF fbDirCreate4.udiStatus < 65534 THEN
					eStatus		:= Error;

					IF fbDirCreate4.udiStatus = 1908 THEN
						udiStatus	:= 10003;	//Creating LCS Directory Error
					ELSE
						udiStatus	:= fbDirCreate4.udiStatus;
					END_IF
				END_IF

			END_IF

	END_CASE

END_ACTION
```

#### Act_Alarm.st - Do Not Change!!!
```iecst
(** 2019-03-25 **)
ACTION Act_Alarm:

	//Error
	IF EDGEPOS(eStatus = Error) THEN

		tyAlmData.sProgNm		:= p_sProgNm;
		tyAlmData.udiCode		:= udiStatus;
		tyAlmData.eSeverity		:= AlmSeverityError;
		tyAlmData.udiRunTime	:= tyAlmData.udiRunTime + 1;
		tyAlmData.bAlm			:= TRUE;
		tyAlmData.udiModuleNum  := udiModuleNum;
		g_sUsrFolderProgNm		:= p_sProgNm;

		//Get Error Message
		IF tyAlmData.udiCode < 10000 OR tyAlmData.udiCode > 10099 THEN
			tyAlmData.sAlmMsg	:= 'Unknown';
			tyAlmData.sRcyMsg	:= 'Unknown';
		ELSE
			tyAlmData.sAlmMsg	:= a_tyAlmText[tyAlmData.udiCode].sAlmText;
			tyAlmData.sRcyMsg	:= a_tyAlmText[tyAlmData.udiCode].sRcyText;
		END_IF

		sStatTxt	:= tyAlmData.sAlmMsg;

	ELSIF bRstErr AND (tyAlmData.udiCode <> 0) THEN

		tyAlmData.udiCode	:= 0;
		tyAlmData.eSeverity	:= AlmSeverityNA;
		tyAlmData.sAlmMsg	:= '';
		tyAlmData.sRcyMsg	:= '';
		tyAlmData.bAlm		:= FALSE;

		sStatTxt	:= a_sStatText[eStat];

	END_IF

END_ACTION
```

#### InputRef.var - Do Not Change!!!
```iecst
(*2019-03-25*)
(**)
(*General*)
VAR
	p_eAct : REFERENCE TO eUsrFolderAction;
	p_udiRstErr : REFERENCE TO UDINT;
	p_sProgNm : REFERENCE TO STRING[15];
END_VAR
```

#### Local.var - Do Not Change!!!
```iecst
(*2019-05-09*)
(**)
(*Local Action, State & Status*)
VAR
	eAct : eUsrFolderAction := UsrFolderActIdle;
	eStat : eUsrFolderAction := UsrFolderActIdle;
	eStatus : eFBStatus := Idle;
	udiStatus : UDINT := 0;
	sStatTxt : STRING[200] := '';
	a_sStatText : ARRAY[0..50] OF STRING[200] := ['Idling','Creating User Directory','Creating Private Directory','Creating Log Directory','Creating LCS Directory',46('')];
END_VAR
(**)
(*Local Alarm*)
VAR
	tyAlmData : tyAlmDat;
	a_tyAlmText : ARRAY[10000..10099] OF tyAlmTxt := [(sAlmText:='Creating User Directory Error',sRcyText:='An Error Occured While Attempting To Create User Directory. Please Contact Nutek For A Possible Solution'),(sAlmText:='Creating Private Directory Error',sRcyText:='An Error Occured While Attempting To Create Private Directory. Please Contact Nutek For A Possible Solution'),(sAlmText:='Creating Log Directory Error',sRcyText:='An Error Occured While Attempting To Create Log Directory. Please Contact Nutek For A Possible Solution'),(sAlmText:='Creating LCS Directory Error',sRcyText:='An Error Occured While Attempting To Create LCS Directory. Please Contact Nutek For A Possible Solution'),96(0)];
END_VAR
(**)
(*Local Output*)
(**)
(*Local Input*)
VAR
	udiRstErr : UDINT := 0;
	sProgNm : STRING[15] := 'UsrFolder';
END_VAR
(**)
(*Local*)
VAR
	bRstErr : BOOL;
	udiRstErrOld : UDINT;
	bInitDone : BOOL;
	bInitialDone : BOOL;
	fbDirCreate1 : fbDirCreate;
	fbDirCreate2 : fbDirCreate;
	fbDirCreate3 : fbDirCreate;
	fbDirCreate4 : fbDirCreate;
END_VAR
(**)
VAR
	udiModuleNum : UDINT := 5551;
END_VAR
```

### LibVer.var - Change By Project
```iecst
(*2019-03-25*)
(**)
(*Action & State & Status*)
VAR
	p_LibVerStat : UDINT;
	p_LibVerStatus : UDINT;
	p_LibVerStatTxt : UDINT;
END_VAR
(**)
(*Alarm*)
VAR
	p_LibVerAlmData : UDINT;
END_VAR
(**)
(*Output*)
VAR
	p_LibVerInfoOut : UDINT;
	p_VerMismatch : UDINT;
END_VAR
```

### LibVer.typ - Do Not Change!!!
```iecst
(*2018-12-07*)
(**)
(*Action*)

TYPE
	eLibVerAction :
		(
		LibVerActIdle,
		LibVerActCreateDir,
		LibVerActWrite,
		LibVerActRead,
		LibVerActReadChk
		);
END_TYPE
```

### Program Logical/LibVer/LibVer (IEC) - 1.00.0 - NtVersion v5.00.0 , NtFileIO v5.00.0

#### InputRef.var
```iecst
(*2019-03-25*)
(**)
(*General*)
VAR
	p_eAct : REFERENCE TO eLibVerAction;
	p_udiRstErr : REFERENCE TO UDINT;
END_VAR
(**)
(*Configuration*)
VAR
	pa_tyInfoIn : REFERENCE TO ARRAY[0..c_diLibNum] OF tyLibrariesVer;
	p_sProgNm : REFERENCE TO STRING[15];
	p_bNtSettingsLoadDone : REFERENCE TO BOOL;
END_VAR
```

#### Local.var
```iecst
(*2020-08-17*)
(**)
(*Local Action, State & Status*)
VAR
	eAct : eLibVerAction := LibVerActIdle;
	eStat : eLibVerAction := LibVerActIdle;
	eStatus : eFBStatus := Idle;
	udiStatus : UDINT := 0;
	sStatTxt : STRING[200] := '';
	a_sStatText : ARRAY[0..50] OF STRING[200] := ['Idling','Creating Directory','Writing Files','Reading Files','Checking Version',46('')];
END_VAR
(**)
(*Local Alarm*)
VAR
	tyAlmData : tyAlmDat;
	a_tyAlmText : ARRAY[10000..10099] OF tyAlmTxt := [(sAlmText:='Creating Private Directory Error',sRcyText:='An Error Occurred While Attempting To Create Private Directory. Please Contact Nutek For A Possible Solution'),(sAlmText:='Creating User Management Directory Error',sRcyText:='An Error Occurred While Attempting To Create User Management Directory. Please Contact Nutek For A Possible Solution'),(sAlmText:='File Open Error While Writing',sRcyText:='An Error Was Encountered While Trying To Open File. Please Contact Nutek For A Possible Solution.'),(sAlmText:='File Create Error While Writing',sRcyText:='An Error Was Encountered While Trying To Create File. Please Contact Nutek For A Possible Solution.'),(sAlmText:='File Write Error',sRcyText:='An Error Was Encountered While Trying To Write File. Please Contact Nutek For A Possible Solution.'),(sAlmText:='File Close Error While Writing',sRcyText:='An Error Was Encountered While Trying To Close File. Please Contact Nutek For A Possible Solution.'),(sAlmText:='File Open Error While Reading',sRcyText:='An Error Was Encountered While Trying To Open File. Please Contact Nutek For A Possible Solution.'),(sAlmText:='File Read Error',sRcyText:='An Error Was Encountered While Trying To Read File. Please Contact Nutek For A Possible Solution.'),(sAlmText:='File Close Error While Reading',sRcyText:='An Error Was Encountered While Trying To Close File. Please Contact Nutek For A Possible Solution.'),(sAlmText:='File Open Error While Checking',sRcyText:='An Error Was Encountered While Trying To Open File. Please Contact Nutek For A Possible Solution.'),(sAlmText:='File Read Error While Checking',sRcyText:='An Error Was Encountered While Trying To Read File. Please Contact Nutek For A Possible Solution.'),(sAlmText:='File Close Error While Checking',sRcyText:='An Error Was Encountered While Trying To Close File. Please Contact Nutek For A Possible Solution.'),(sAlmText:='Libraries Version Mismatch',sRcyText:='Libraries Version Mismatch. Please Contact Nutek For A Possible Solution.'),(sAlmText:='Directory Does Not Exist While Writing',sRcyText:='The Directory Does Not Exist. Please Contact Nutek For A Possible Solution.'),(sAlmText:='File Not Found While Reading',sRcyText:='File Not Found. Please Contact Nutek For A Possible Solution.'),(sAlmText:='File Not Found While Checking',sRcyText:='File Not Found. Please Contact Nutek For A Possible Solution.'),(sAlmText:='Libraries Version File Check Error',sRcyText:='Libraries Files Corrupted. Please Contact Nutek For A Possible Solution.'),83((0))];
END_VAR
(**)
(*Local Output*)
VAR
	a_tyInfoOut : ARRAY[0..c_diLibNum] OF tyLibrariesVer;
	a_bVerMismatch : ARRAY[0..c_diLibNum] OF BOOL;
END_VAR
(**)
(*Local Input*)
VAR
	udiRstErr : UDINT := 0;
	a_tyInfoIn : ARRAY[0..c_diLibNum] OF tyLibrariesVer;
	sProgNm : STRING[15] := 'LibVer';
	bNtSettingsLoadDone : BOOL := TRUE;
END_VAR
(**)
(*Local*)
VAR
	bRstErr : BOOL;
	udiRstErrOld : UDINT;
	bInitDone : BOOL;
	bInitialDone : BOOL;
	usiStep : USINT;
	di : DINT;
	fbDirCreate1 : fbDirCreate;
	fbDirCreate2 : fbDirCreate;
	fbFileRead1 : fbFileFullRead;
	fbFileWrite1 : fbFileFullWrite;
	fbChkLibVerFile : fbChkFileValidity;
	fbChkLibVer : fbChkLibrariesVer;
	udiModuleNum : UDINT := 5451;
END_VAR
```

#### Act_Action.st
```iecst
(** 2019-03-25 **)
ACTION Act_Action:

	//Reset Error
	IF (eStatus = Error) AND bRstErr THEN
		p_eAct	:= LibVerActIdle;
		eStat	:= LibVerActIdle;
	END_IF

	//Reset Done
	IF eStatus = Done AND p_eAct = LibVerActIdle THEN
		eStat	:= LibVerActIdle;
	END_IF

	//Set p_eAct
	IF eStatus = Idle THEN
		eStat	:= p_eAct;
	END_IF

END_ACTION
```

#### Act_Alarm.st
```iecst
(** 2022-12-20 **)
ACTION Act_Alarm:

	//Error
	IF EDGEPOS(eStatus = Error) THEN

		tyAlmData.sProgNm		:= p_sProgNm;
		tyAlmData.udiCode		:= udiStatus;
		tyAlmData.udiRunTime	:= tyAlmData.udiRunTime + 1;

		tyAlmData.udiModuleNum  := udiModuleNum;
		g_sLibVerProgNm			:= p_sProgNm;

		IF tyAlmData.udiCode = 10012 THEN
			tyAlmData.eSeverity	:= AlmSeverityWarning;
			tyAlmData.bWarning		:= TRUE;
			//Get Error Message
			tyAlmData.sAlmMsg	:= a_tyAlmText[tyAlmData.udiCode].sAlmText;

			FOR di := 0 TO c_diLibNum DO
				IF a_bVerMismatch[di] = TRUE THEN
					tyAlmData.sAlmMsg	:= CONCAT(tyAlmData.sAlmMsg , ' (');
					tyAlmData.sAlmMsg	:= CONCAT(tyAlmData.sAlmMsg , a_tyInfoOut[di].sName);
					tyAlmData.sAlmMsg	:= CONCAT(tyAlmData.sAlmMsg , ')');
					g_sLiberWarnName    := a_tyInfoOut[di].sName;
					EXIT;
				END_IF
			END_FOR

			tyAlmData.sRcyMsg	:= a_tyAlmText[tyAlmData.udiCode].sRcyText;

		ELSE
			tyAlmData.eSeverity	:= AlmSeverityError;
			tyAlmData.bAlm			:= TRUE;
			//Get Error Message
			IF tyAlmData.udiCode < 10000 OR tyAlmData.udiCode > 10099 THEN
				tyAlmData.sAlmMsg	:= 'Unknown';
				tyAlmData.sRcyMsg	:= 'Unknown';
			ELSE
				tyAlmData.sAlmMsg	:= a_tyAlmText[tyAlmData.udiCode].sAlmText;
				tyAlmData.sRcyMsg	:= a_tyAlmText[tyAlmData.udiCode].sRcyText;
			END_IF

			sStatTxt	:= tyAlmData.sAlmMsg;

		END_IF

	ELSIF bRstErr AND (tyAlmData.udiCode <> 0) THEN

		tyAlmData.udiCode	:= 0;
		tyAlmData.eSeverity	:= AlmSeverityNA;
		tyAlmData.sAlmMsg	:= '';
		tyAlmData.sRcyMsg	:= '';
		tyAlmData.bAlm			:= FALSE;
		tyAlmData.bWarning		:= FALSE;
		sStatTxt	:= a_sStatText[eStat];

	END_IF

END_ACTION
```

#### Act_InitGlobal.st
```iecst
(** 2019-03-25 **)
ACTION Act_InitGlobal:

	(* Always Change If Project Change *)

	//Pass Data To Link

	//Pass Data To Internal Use
	p_udiRstErr ACCESS p_RstErrReset;
	p_eAct ACCESS p_StartupLibVerAct;
	p_sProgNm ACCESS p_NtParamLibVersionProgNm;
	p_bNtSettingsLoadDone ACCESS p_StartupNtSettingsLoadDone;

	(* Always Change If Project Change *)

END_ACTION
```

#### Act_Initial.st
```iecst
(** 2020-08-17 **)
ACTION Act_Initial:

	//Initial
	sStatTxt	:= a_sStatText[eStat];

	fbDirCreate1.sDevice	:= 'F';
	fbDirCreate1.sDirName	:= 'User';
	fbDirCreate1(bEn := FALSE);

	fbDirCreate2.sDevice	:= 'User';
	fbDirCreate2.sDirName	:= 'LibrariesVersion';
	fbDirCreate2(bEn := FALSE);

	fbFileRead1.sDevice		:= 'LibVer';
	fbFileRead1.sFile		:= 'LibrariesVersion.dat';
	fbFileRead1.udiOffset	:= 0;
	fbFileRead1.p_Dest		:= ADR(a_tyInfoOut);
	fbFileRead1.udiLen		:= SIZEOF(a_tyInfoOut);
	fbFileRead1(bEn := FALSE);

	fbFileWrite1.sDevice	:= 'LibVer';
	fbFileWrite1.sFile		:= 'LibrariesVersion.dat';
	fbFileWrite1.udiOffset	:= 0;
	fbFileWrite1.p_Src		:= ADR(pa_tyInfoIn);
	fbFileWrite1.udiLen		:= SIZEOF(pa_tyInfoIn);
	fbFileWrite1.udiOption	:= 0;
	fbFileWrite1(bEn := FALSE);

	fbChkLibVerFile(bEn := FALSE);

	fbChkLibVer.pa_bVerMismatch := ADR(a_bVerMismatch);
	fbChkLibVer(bEn := FALSE);

END_ACTION
```

#### Act_InitLocal.st
```iecst
(** 2019-03-25 **)
ACTION Act_InitLocal:

	//Input Reference Link To Local Variable
	p_eAct ACCESS ADR(eAct);
	p_udiRstErr ACCESS ADR(udiRstErr);
	pa_tyInfoIn ACCESS ADR(a_tyInfoIn);
	p_sProgNm ACCESS ADR(sProgNm);
	p_bNtSettingsLoadDone ACCESS ADR(bNtSettingsLoadDone);

END_ACTION
```

#### Act_Main.st
```iecst
(** 2020-08-17 **)
ACTION Act_Main:

	//Main
	CASE eStat OF

		LibVerActIdle:
			IF eStatus <> Idle THEN	//Reset Data
				//Private
				fbDirCreate1(bEn := FALSE);
				fbDirCreate2(bEn := FALSE);
				fbFileRead1(bEn := FALSE);
				fbFileWrite1(bEn := FALSE);
				fbChkLibVerFile(bEn := FALSE);
				fbChkLibVer(bEn := FALSE);
				usiStep	:= 0;
				memset(ADR(a_bVerMismatch), 0, SIZEOF(a_bVerMismatch));

				sStatTxt	:= a_sStatText[eStat];

			END_IF

			eStatus	:= Idle;

		LibVerActCreateDir:
			IF eStatus = Idle OR eStatus = Busy THEN

				eStatus	:= Busy;

				sStatTxt	:= a_sStatText[eStat];

				CASE usiStep OF
					0:
						fbDirCreate1(bEn := TRUE);
						IF fbDirCreate1.udiStatus = 0 THEN
							usiStep	:= 1;
						ELSIF fbDirCreate1.udiStatus < 65534 THEN
							eStatus		:= Error;

							IF fbDirCreate1.udiStatus = 1908 THEN
								udiStatus	:= 10000;	//Creating Private Directory Error
							ELSE
								udiStatus	:= fbDirCreate1.udiStatus;
							END_IF
						END_IF

					1:
						fbDirCreate2(bEn := TRUE);
						IF fbDirCreate2.udiStatus = 0 THEN
							eStatus	:= Done;
						ELSIF fbDirCreate2.udiStatus < 65534 THEN
							eStatus		:= Error;

							IF fbDirCreate2.udiStatus = 1908 THEN
								udiStatus	:= 10001;	//Creating User Management Directory Error
							ELSE
								udiStatus	:= fbDirCreate2.udiStatus;
							END_IF
						END_IF

				END_CASE

			END_IF

		LibVerActWrite:
			IF eStatus = Idle OR eStatus = Busy THEN

				eStatus	:= Busy;

				sStatTxt	:= a_sStatText[eStat];

				fbFileWrite1(bEn := TRUE);

				IF fbFileWrite1.udiStatus = 0 THEN
					eStatus	:= Done;
				ELSIF fbFileWrite1.udiStatus < 65534 THEN
					eStatus			:= Error;

					IF fbFileWrite1.udiStatus = 1900 THEN
						udiStatus	:= 10002;	//File Open Error While Writing
					ELSIF fbFileWrite1.udiStatus = 1901 THEN
						udiStatus	:= 10003;	//File Create Error While Writing
					ELSIF fbFileWrite1.udiStatus = 1903 THEN
						udiStatus	:= 10004;	//File Write Error
					ELSIF fbFileWrite1.udiStatus = 1904 THEN
						udiStatus	:= 10005;	//File Close Error While Writing
					ELSIF fbFileWrite1.udiStatus = 1914 THEN
						udiStatus	:= 10013;	//Directory Does Not Exist While Writing
					ELSE
						udiStatus	:= fbFileWrite1.udiStatus;
					END_IF
				END_IF

			END_IF

		LibVerActRead:
			IF eStatus = Idle OR eStatus = Busy THEN

				eStatus	:= Busy;

				sStatTxt	:= a_sStatText[eStat];

				fbFileRead1(bEn := TRUE);
				IF fbFileRead1.udiStatus = 0 THEN
					eStatus	:= Done;
				ELSIF fbFileRead1.udiStatus < 65534 THEN
					eStatus		:= Error;

					IF fbFileRead1.udiStatus = 1900 THEN
						udiStatus	:= 10006;	//File Open Error While Reading
					ELSIF fbFileRead1.udiStatus = 1902 THEN
						udiStatus	:= 10007;	//File Read Error
					ELSIF fbFileRead1.udiStatus = 1904 THEN
						udiStatus	:= 10008;	//File Close Error While Reading
					ELSIF fbFileRead1.udiStatus = 1915 THEN
						udiStatus	:= 10014;	//File Not Found While Reading
					ELSE
						udiStatus	:= fbFileRead1.udiStatus;
					END_IF
				END_IF

			END_IF

		LibVerActReadChk:
			IF eStatus = Idle OR eStatus = Busy THEN

				eStatus	:= Busy;

				sStatTxt	:= a_sStatText[eStat];

				CASE usiStep OF
					0:
						fbFileRead1(bEn := TRUE);
						IF fbFileRead1.udiStatus = 0 THEN
							usiStep	:= 1;
						ELSIF fbFileRead1.udiStatus < 65534 THEN
							eStatus		:= Error;

							IF fbFileRead1.udiStatus = 1900 THEN
								udiStatus	:= 10009;	//File Open Error While Checking
							ELSIF fbFileRead1.udiStatus = 1902 THEN
								udiStatus	:= 10010;	//File Read Error While Checking
							ELSIF fbFileRead1.udiStatus = 1904 THEN
								udiStatus	:= 10011;	//File Close Error While Checking
							ELSIF fbFileRead1.udiStatus = 1915 THEN
								udiStatus	:= 10015;	//File Not Found While Checking
							ELSE
								udiStatus	:= fbFileRead1.udiStatus;
							END_IF
						END_IF

					1:
						fbChkLibVerFile.a_tyLibraryVer := a_tyInfoOut;

						fbChkLibVerFile(bEn := TRUE);
						IF fbChkLibVerFile.udiStatus = 0 THEN
							usiStep	:= 2;
						ELSIF fbChkLibVerFile.udiStatus < 65534 THEN
							eStatus		:= Error;

							IF fbChkLibVerFile.udiStatus = 1001 THEN
								udiStatus	:= 10016;	//Libraries Version File Corrupted
							END_IF
						END_IF

					2:

						fbChkLibVer.a_tyLibraryVer := a_tyInfoOut;

						fbChkLibVer(bEn := TRUE);
						IF fbChkLibVer.udiStatus = 0 THEN
							eStatus	:= Done;
						ELSIF fbChkLibVer.udiStatus < 65534 THEN
							eStatus		:= Error;

							IF fbChkLibVer.udiStatus = 1002 THEN
								udiStatus	:= 10012;	//Libraries Version Mismatch
							END_IF
						END_IF

				END_CASE

			END_IF

	END_CASE

END_ACTION
```

#### Init.st
```iecst
(** 2019-03-25 **)
PROGRAM _INIT

	(* Always Change If Project Change *)

	//Pass Address To Global Address For External Use
	//Action, State & Status
	p_LibVerStat	:= ADR(eStat);
	p_LibVerStatus	:= ADR(eStatus);
	p_LibVerStatTxt	:= ADR(sStatTxt);

	//Alarm
	p_LibVerAlmData	:= ADR(tyAlmData);

	//Output
	p_LibVerInfoOut	:= ADR(a_tyInfoOut);
	p_VerMismatch	:= ADR(a_bVerMismatch);

	(* Always Change If Project Change *)

END_PROGRAM
```

### Time.var - Change By Project
```iecst
(*2019-03-25*)
(**)
(*Action & State & Status*)
VAR
	p_TimeStat : UDINT;
	p_TimeStatus : UDINT;
	p_TimeStatTxt : UDINT;
END_VAR
(**)
(*Alarm*)
VAR
	p_TimeAlmData : UDINT;
	p_TimeAlmData1 : UDINT;
END_VAR
(**)
(*Output*)
VAR
	p_TimeCurrDT : UDINT;
	p_TimeCurrTimeZone : UDINT;
	p_TimeCurrDTStruct : UDINT;
END_VAR
```

### Time.typ - Do Not Change!!!
```iecst
(*2018-12-07*)
(**)
(*Action*)

TYPE
	eTimeAction :
		(
		TimeActIdle,
		TimeActGetTime,
		TimeActGetTimeZone,
		TimeActSetTime,
		TimeActSetTimeZone
		);
END_TYPE
```

### Program Logical/Time/Time (IEC, version 1.00.0) - 1.00.0 - (2018-12-07)

#### Init.st - Change By Project
```iecst
(** 2019-03-25 **)
PROGRAM _INIT

	(* Always Change If Project Change *)

	//Pass Address To Global Address For External Use
	//Action, State & Status
	p_TimeStat		:= ADR(eStat);
	p_TimeStatus	:= ADR(eMainStatus);
	p_TimeStatTxt	:= ADR(sStatTxt);

	//Alarm
	p_TimeAlmData	:= ADR(tyAlmData);
	p_TimeAlmData1	:= ADR(tyAlmData1);

	//Output
	p_TimeCurrDT		:= ADR(dtCurrDT);
	p_TimeCurrTimeZone	:= ADR(uiCurrTimeZone);
	p_TimeCurrDTStruct	:= ADR(tyCurrDTStruct);

	(* Always Change If Project Change *)

END_PROGRAM
```

#### Act_InitGlobal.st - Change By Project
```iecst
(** 2019-05-22 **)
ACTION Act_InitGlobal:

	(* Always Change If Project Change *)

	//Pass Data To Link

	//Pass Data To Internal Use
	p_eAct ACCESS p_LFFollowerTimeAct;
	p_udiRstErr ACCESS p_RstErrReset;
	p_dtSetDT ACCESS p_LFFollowerSetDT;
	p_sProgNm ACCESS p_NtParamTimeProgNm;
	p_bNtSettingsLoadDone ACCESS p_StartupNtSettingsLoadDone;

	(* Always Change If Project Change *)

END_ACTION
```

#### Cyclic.st - Do Not Change!!!
```iecst
(** 2019-03-29 **)
PROGRAM _CYCLIC

	IF bInitDone = FALSE THEN
		bInitDone	:= TRUE;

		Act_InitLocal;
		Act_InitGlobal;

	ELSIF bInitialDone = FALSE THEN
		IF p_bNtSettingsLoadDone = TRUE THEN
			bInitialDone	:= TRUE;

			Act_Initial;
		END_IF

	ELSE

		Act_Background;
		Act_RstErr;
		Act_LinkAction;
		Act_Action;
		Act_Link;
		Act_Main;
		Act_CombineErr;
		Act_Alarm;
		Act_Alarm1;

	END_IF

END_PROGRAM
```

#### Act_InitLocal.st - Do Not Change!!!
```iecst
(** 2019-03-25 **)
ACTION Act_InitLocal:

	//Input Reference Link To Local Variable
	p_eAct ACCESS ADR(eAct);
	p_udiRstErr ACCESS ADR(udiRstErr);
	p_dtSetDT ACCESS ADR(dtSetDT);
	p_uiSetTimeZone ACCESS ADR(uiSetTimeZone);
	p_sProgNm ACCESS ADR(sProgNm);
	p_bNtSettingsLoadDone ACCESS ADR(bNtSettingsLoadDone);

END_ACTION
```

#### Act_Initial.st - Do Not Change!!!
```iecst
(** 2019-01-03 **)
ACTION Act_Initial:

	//Initial
	sStatTxt	:= a_sStatText[eStat];

	fbSetTime(enable := FALSE);

	fbSetTimeZone.option	:= cfgOPTION_NON_VOLATILE;
	fbSetTimeZone(enable := FALSE);

	fbGetTime(enable := FALSE);

	fbGetTime1(enable := FALSE);

	fbGetTimeDT.pDTStructure	:= ADR(tyCurrDTStruct);
	fbGetTimeDT(enable := FALSE);

	fbGetTimeDT1.pDTStructure	:= ADR(tyCurrDTStruct);
	fbGetTimeDT1(enable := FALSE);

	fbGetTimeZone(enable := FALSE);

	fbDlyTm(IN := FALSE);

END_ACTION
```

#### Act_Action.st - Do Not Change!!!
```iecst
(** 2019-03-25 **)
ACTION Act_Action:

	//Reset Error
	IF (eStatus = Error) AND bRstErr THEN
		p_eAct	:= TimeActIdle;
		eStat	:= TimeActIdle;
	END_IF

	//Reset Done
	IF eStatus = Done AND p_eAct = TimeActIdle THEN
		eStat	:= TimeActIdle;
	END_IF

	//Set p_eAct
	IF eStatus = Idle THEN
		eStat	:= p_eAct;
	END_IF

END_ACTION
```

#### Act_Main.st - Do Not Change!!!
```iecst
(** 2019-01-02 **)
ACTION Act_Main:

	//Main
	CASE eStat OF

		TimeActIdle:
			IF eStatus <> Idle THEN	//Reset Data
				//Private
				fbSetTime(enable := FALSE);
				fbSetTimeZone(enable := FALSE);
				fbGetTime(enable := FALSE);
				fbGetTimeDT(enable := FALSE);
				fbGetTimeZone(enable := FALSE);

				sStatTxt	:= a_sStatText[eStat];

			END_IF

			eStatus	:= Idle;

		TimeActSetTime:
			IF eStatus = Idle OR eStatus = Busy THEN

				eStatus	:= Busy;

				sStatTxt	:= a_sStatText[eStat];

				fbSetTime.DT1	:= p_dtSetDT;
				fbSetTime(enable := TRUE);

				IF fbSetTime.status = 0 THEN
					eStatus	:= Done;
				ELSIF fbSetTime.status < 65534 THEN
					udiStatus	:= 10000;	//Set Time Error
					eStatus		:= Error;
				END_IF

			END_IF

		TimeActSetTimeZone:
			IF eStatus = Idle OR eStatus = Busy THEN

				eStatus	:= Busy;

				sStatTxt	:= a_sStatText[eStat];

				fbSetTimeZone.timezoneID	:= p_uiSetTimeZone;
				fbSetTimeZone(enable := TRUE);

				IF fbSetTimeZone.status = 0 THEN
					eStatus	:= Done;
				ELSIF fbSetTimeZone.status < 65534 THEN
					udiStatus	:= 10001;	//Set Time Zone Error
					eStatus		:= Error;
				END_IF

			END_IF

		TimeActGetTime:
			IF eStatus = Idle OR eStatus = Busy THEN

				eStatus	:= Busy;

				sStatTxt	:= a_sStatText[eStat];

				fbGetTime(enable := TRUE);
				fbGetTimeDT(enable := TRUE);

				IF fbGetTime.status = 0 AND fbGetTimeDT.status = 0 THEN
					dtCurrDT	:= fbGetTime.DT1;
					eStatus		:= Done;
				ELSIF fbGetTime.status > 0 AND fbGetTime.status < 65534 THEN
					udiStatus	:= 10002;	//Get Time Error
					eStatus		:= Error;
				ELSIF fbGetTimeDT.status > 0 AND fbGetTimeDT.status < 65534 THEN
					udiStatus	:= 10003;	//Get Time Structure Error
					eStatus		:= Error;
				END_IF

			END_IF

		TimeActGetTimeZone:
			IF eStatus = Idle OR eStatus = Busy THEN

				eStatus	:= Busy;

				sStatTxt	:= a_sStatText[eStat];

				fbGetTimeZone(enable := TRUE);

				IF fbGetTimeZone.status = 0 THEN
					uiCurrTimeZone	:= fbGetTimeZone.timezoneID;
					eStatus			:= Done;
				ELSIF fbGetTimeZone.status < 65534 THEN
					udiStatus	:= 10004;	//Get Time Zone Error
					eStatus		:= Error;
				END_IF

			END_IF

	END_CASE

END_ACTION
```

#### Act_Background.st - Do Not Change!!!
```iecst
(** 2019-01-21 **)
ACTION Act_Background:

	IF (eStatus1 = Error) AND bRstErr THEN
		eStatus1	:= Idle;
		udiStatus1	:= 0;
		fbDlyTm(IN := FALSE);
		fbGetTime1(enable := FALSE);
		fbGetTimeDT1(enable := FALSE);
	END_IF

	IF eStatus1 <> Error THEN

		fbDlyTm(IN := TRUE);

		IF fbDlyTm.Q = TRUE THEN

			fbGetTime1(enable := TRUE);
			fbGetTimeDT1(enable := TRUE);

			IF fbGetTime1.status = 0 AND fbGetTimeDT1.status = 0 THEN
				dtCurrDT	:= fbGetTime1.DT1;
				fbGetTime1(enable := FALSE);
				fbGetTimeDT1(enable := FALSE);
				fbDlyTm(IN := FALSE);
			ELSIF fbGetTime1.status > 0 AND fbGetTime1.status < 65534 THEN
				udiStatus1	:= 10005;	//Get Time Error In Background
				eStatus1	:= Error;
			ELSIF fbGetTimeDT1.status > 0 AND fbGetTimeDT1.status < 65534 THEN
				udiStatus1	:= 10006;	//Get Time Structure Error In Background
				eStatus1	:= Error;
			END_IF

		END_IF

	END_IF

END_ACTION
```

#### Act_CombineErr.st - Do Not Change!!!
```iecst
(** 2019-01-21 **)
ACTION Act_CombineErr:

	//Combine Error
	IF eStatus = Error OR eStatus1 = Error THEN
		eMainStatus	:= Error;
	ELSE
		eMainStatus	:= eStatus;
	END_IF

END_ACTION
```

#### Act_Alarm.st - Do Not Change!!!
```iecst
(** 2019-03-25 **)
ACTION Act_Alarm:

	//Error
	IF EDGEPOS(eStatus = Error) THEN

		tyAlmData.sProgNm		:= p_sProgNm;
		tyAlmData.udiCode		:= udiStatus;
		tyAlmData.eSeverity		:= AlmSeverityError;
		tyAlmData.udiRunTime	:= tyAlmData.udiRunTime + 1;
		tyAlmData.bAlm			:= TRUE;
		tyAlmData.udiModuleNum  := udiModuleNum;
		g_sTimeProgNm			:= p_sProgNm;

		//Get Error Message
		IF tyAlmData.udiCode < 10000 OR tyAlmData.udiCode > 10099 THEN
			tyAlmData.sAlmMsg	:= 'Unknown';
			tyAlmData.sRcyMsg	:= 'Unknown';
		ELSE
			tyAlmData.sAlmMsg	:= a_tyAlmText[tyAlmData.udiCode].sAlmText;
			tyAlmData.sRcyMsg	:= a_tyAlmText[tyAlmData.udiCode].sRcyText;
		END_IF

		sStatTxt	:= tyAlmData.sAlmMsg;

	ELSIF bRstErr AND (tyAlmData.udiCode <> 0) THEN

		tyAlmData.udiCode	:= 0;
		tyAlmData.eSeverity	:= AlmSeverityNA;
		tyAlmData.sAlmMsg	:= '';
		tyAlmData.sRcyMsg	:= '';
		tyAlmData.bAlm			:= FALSE;

		sStatTxt	:= a_sStatText[eStat];

	END_IF

END_ACTION
```

#### Act_Alarm1.st - Do Not Change!!!
```iecst
(** 2019-03-25 **)
ACTION Act_Alarm1:

	//Error
	IF EDGEPOS(eStatus1 = Error) THEN

		tyAlmData1.sProgNm		:= p_sProgNm;
		tyAlmData1.udiCode		:= udiStatus1;
		tyAlmData1.eSeverity	:= AlmSeverityError;
		tyAlmData1.udiRunTime	:= tyAlmData1.udiRunTime + 1;
		tyAlmData1.bAlm			:= TRUE;
		tyAlmData1.udiModuleNum  := udiModuleNum;
		g_sTimeProgNm			:= p_sProgNm;

		//Get Error Message
		IF tyAlmData1.udiCode < 10000 OR tyAlmData1.udiCode > 10099 THEN
			tyAlmData1.sAlmMsg	:= 'Unknown';
			tyAlmData1.sRcyMsg	:= 'Unknown';
		ELSE
			tyAlmData1.sAlmMsg	:= a_tyAlmText[tyAlmData1.udiCode].sAlmText;
			tyAlmData1.sRcyMsg	:= a_tyAlmText[tyAlmData1.udiCode].sRcyText;
		END_IF

		sStatTxt	:= tyAlmData1.sAlmMsg;

	ELSIF bRstErr AND (tyAlmData1.udiCode <> 0) THEN

		tyAlmData1.udiCode		:= 0;
		tyAlmData1.eSeverity	:= AlmSeverityNA;
		tyAlmData1.sAlmMsg		:= '';
		tyAlmData1.sRcyMsg		:= '';
		tyAlmData1.bAlm			:= FALSE;

		sStatTxt	:= a_sStatText[eStat];

	END_IF

END_ACTION
```

#### InputRef.var - Do Not Change!!!
```iecst
(*2019-03-25*)
(**)
(*General*)
VAR
	p_eAct : REFERENCE TO eTimeAction;
	p_udiRstErr : REFERENCE TO UDINT;
END_VAR
(**)
(*Configuration*)
VAR
	p_dtSetDT : REFERENCE TO DATE_AND_TIME;
	p_uiSetTimeZone : REFERENCE TO UINT;
	p_sProgNm : REFERENCE TO STRING[15];
	p_bNtSettingsLoadDone : REFERENCE TO BOOL;
END_VAR
```

#### Local.var - Do Not Change!!!
```iecst
(*2019-04-30*)
(**)
(*Local Action, State & Status*)
VAR
	eAct : eTimeAction := TimeActIdle;
	eStat : eTimeAction := TimeActIdle;
	eMainStatus : eFBStatus := Idle;
	eStatus : eFBStatus := Idle;
	eStatus1 : eFBStatus := Idle;
	udiStatus : UDINT := 0;
	udiStatus1 : UDINT := 0;
	sStatTxt : STRING[200] := '';
	a_sStatText : ARRAY[0..50] OF STRING[200] := ['Idling','Get Time','Get Time Zone','Setting Time','Setting Time Zone',46('')];
END_VAR
(**)
(*Local Alarm*)
VAR
	tyAlmData : tyAlmDat;
	tyAlmData1 : tyAlmDat;
	a_tyAlmText : ARRAY[10000..10099] OF tyAlmTxt := [(sAlmText:='Set Time Error',sRcyText:='Your Clock Is Set Incorrectly. Please Set Correct Date And Time In Language And Setup.'),(sAlmText:='Set TIME Zone Error',sRcyText:='Invalid TIME Zone. Please Check Your TIME Zone And Try Again.'),(sAlmText:='Get TIME Error',sRcyText:='Getting Invalid Time. Please Set Correct DATE And TIME In Language And Setup.'),(sAlmText:='Get TIME Structure Error',sRcyText:='Invalid TIME Structure. Please Set Correct DATE And TIME In Language And Setup.'),(sAlmText:='Get TIME Zone Error',sRcyText:='Getting Invalid TIME Zone. Please Check Your TIME Zone And Try Again.'),(sAlmText:='Get TIME Error In Background',sRcyText:='Getting Invalid Time. Please Set Correct DATE And TIME In Language And Setup'),(sAlmText:='Get TIME Structure Error In Background',sRcyText:='Invalid TIME Structure. Please Set Correct DATE And TIME In Language And Setup.'),93((0))];
END_VAR
(**)
(*Local Output*)
VAR
	dtCurrDT : DATE_AND_TIME;
	uiCurrTimeZone : UINT;
	tyCurrDTStruct : DTStructure;
END_VAR
(**)
(*Local Input*)
VAR
	udiRstErr : UDINT := 0;
	dtSetDT : DATE_AND_TIME;
	uiSetTimeZone : UINT;
	sProgNm : STRING[15] := 'Time';
	bNtSettingsLoadDone : BOOL := TRUE;
END_VAR
(**)
(*Local*)
VAR
	bRstErr : BOOL;
	udiRstErrOld : UDINT;
	bInitDone : BOOL;
	bInitialDone : BOOL;
	fbDlyTm : TON := (PT:=T#500ms);
	fbGetTime : DTGetTime;
	fbGetTime1 : DTGetTime;
	fbSetTime : DTSetTime;
	fbGetTimeDT : DTStructureGetTime;
	fbGetTimeDT1 : DTStructureGetTime;
	fbGetTimeZone : CfgGetTimeZone;
	fbSetTimeZone : CfgSetTimeZone;
	udiModuleNum : UDINT := 5851;
END_VAR
```

### HWInfo.typ - Do Not Change!!!
```iecst
(*2020-09-22*)
(**)
(*Action*)

TYPE
	eHWInfoAction :
		(
		HWInfoActIdle,
		HWInfoActGetIPAddr,
		HWInfoActGetSubnetMask,
		HWInfoActGetMacAddr,
		HWInfoActSetIPAddr,
		HWInfoActSetSubnetMask,
		HWInfoActGetEthConfigMode,
		HWInfoActSetEthConfigMode
		);
END_TYPE

(**)

TYPE
	eNetworkConfigMod :
		(
		SetIPManually := 0,
		IPFromDHCPServer := 1
		);
END_TYPE
```

### HWInfo.var - Change By Project
```iecst
(*2020-09-22*)
(**)
(*Action & State & Status*)
VAR
	p_HWInfoStat : UDINT;
	p_HWInfoStatus : UDINT;
	p_HWInfoStatTxt : UDINT;
END_VAR
(**)
(*Alarm*)
VAR
	p_HWInfoAlmData : UDINT;
END_VAR
(**)
(*Output*)
VAR
	p_HWInfoIPAddr : UDINT;
	p_HWInfoMacAddr : UDINT;
	p_HWInfoSubnetMask : UDINT;
	p_HWInfoEthMode : UDINT;
END_VAR
```

### Program Logical/HWInfo/HWInfo (IEC) - 1.00.0 - 

#### InputRef.var
```iecst
(*2020-09-22*)
(**)
(*General*)
VAR
	p_eAct : REFERENCE TO eHWInfoAction;
	p_udiRstErr : REFERENCE TO UDINT;
END_VAR
(**)
(*Configuration*)
VAR
	p_sSetIPAddr : REFERENCE TO STRING[15];
	p_sSetSubnetMask : REFERENCE TO STRING[15];
	p_sDevice : REFERENCE TO STRING[3];
	p_sProgNm : REFERENCE TO STRING[15];
	p_usiNetworkMod : REFERENCE TO USINT;
	p_bNtSettingsLoadDone : REFERENCE TO BOOL;
END_VAR
```

#### Local.var
```iecst
(*2020-10-05*)
(**)
(*Local Action, State & Status*)
VAR
	eAct : eHWInfoAction := HWInfoActIdle;
	eStat : eHWInfoAction := HWInfoActIdle;
	eStatus : eFBStatus := Idle;
	udiStatus : UDINT := 0;
	sStatTxt : STRING[200] := '';
	a_sStatText : ARRAY[0..50] OF STRING[200] := ['Idling','Get IP Address','Get IP Subnet Mask','Get Mac Address','Setting IP Address','Setting IP Subnet Mask','Get Ethernet Configuration Mode','Setting Ethernet Configuration Mode',43('')];
END_VAR
(**)
(*Local Alarm*)
VAR
	tyAlmData : tyAlmDat;
	a_tyAlmText : ARRAY[10000..10099] OF tyAlmTxt := [(sAlmText:='Get IP Address Error',sRcyText:='Failed To Obtain The IP Address. Please Contact Nutek For A Possible Solution.'),(sAlmText:='Get Subnet Mask Error',sRcyText:='Failed To Obtain The Subnet Mask. Please Contact Nutek For A Possible Solution.'),(sAlmText:='Get Mac Address Error',sRcyText:='Failed To Obtain The Mac Address. Please Contact Nutek For A Possible Solution.'),(sAlmText:='Set IP Address Error',sRcyText:='Invalid IP Address Configuration. Please Contact Nutek For A Possible Solution.'),(sAlmText:='Set Subnet Mask Error',sRcyText:='Invalid Subnet Mask Configuration. Please Contact Nutek For A Possible Solution.'),(sAlmText:='Get Network Configuration Mode Error',sRcyText:='Failed To Obtain The Network Configuration. Please Contact Nutek For A Possible Solution.'),(sAlmText:='Set Network Configuration Mode Error',sRcyText:='Invalid Network Configuration . Please Contact Nutek For A Possible Solution.'),93(0)];
END_VAR
(**)
(*Local Output*)
VAR
	sIPAddr : STRING[15];
	sSubnetMask : STRING[15];
	a_usiMacAddr : ARRAY[0..5] OF USINT;
	udiConfigMode : UDINT;
END_VAR
(**)
(*Local Input*)
VAR
	udiRstErr : UDINT := 0;
	sSetIPAddr : STRING[15];
	sSetSubnetMask : STRING[15];
	sDevice : STRING[3] := 'IF2';
	sProgNm : STRING[15] := 'HWInfo';
	bNtSettingsLoadDone : BOOL := TRUE;
	usiNetworkMode : USINT;
END_VAR
(**)
(*Local*)
VAR
	bRstErr : BOOL;
	udiRstErrOld : UDINT;
	bInitDone : BOOL;
	bInitialDone : BOOL;
	fbGetIPAddr : CfgGetIPAddr;
	fbGetSubnetMask : CfgGetSubnetMask;
	fbGetMacAddr : CfgGetMacAddr;
	fbSetIPAddr : CfgSetIPAddr;
	fbSetSubnetMask : CfgSetSubnetMask;
	fbSetETHConfigMode : CfgSetEthConfigMode;
	fbGetETHConfigMode : CfgGetEthConfigMode;
	udiModuleNum : UDINT := 5651;
END_VAR
```

#### Act_Action.st
```iecst
(** 2019-03-25 **)
ACTION Act_Action:

	//Reset Error
	IF (eStatus = Error) AND bRstErr THEN
		p_eAct	:= HWInfoActIdle;
		eStat	:= HWInfoActIdle;
	END_IF

	//Reset Done
	IF eStatus = Done AND p_eAct = HWInfoActIdle THEN
		eStat	:= HWInfoActIdle;
	END_IF

	//Set p_eAct
	IF eStatus = Idle THEN
		eStat	:= p_eAct;
	END_IF

END_ACTION
```

#### Act_Alarm.st
```iecst
(** 2019-03-25 **)
ACTION Act_Alarm:

	//Error
	IF EDGEPOS(eStatus = Error) THEN

		tyAlmData.sProgNm		:= p_sProgNm;
		tyAlmData.udiCode		:= udiStatus;
		tyAlmData.eSeverity		:= AlmSeverityError;
		tyAlmData.udiRunTime	:= tyAlmData.udiRunTime + 1;
		tyAlmData.bAlm			:= TRUE;
		tyAlmData.udiModuleNum  := udiModuleNum;
		g_sHWInfoProgNm		:= p_sProgNm;

		//Get Error Message
		IF tyAlmData.udiCode < 10000 OR tyAlmData.udiCode > 10099 THEN
			tyAlmData.sAlmMsg	:= 'Unknown';
			tyAlmData.sRcyMsg	:= 'Unknown';
		ELSE
			tyAlmData.sAlmMsg	:= a_tyAlmText[tyAlmData.udiCode].sAlmText;
			tyAlmData.sRcyMsg	:= a_tyAlmText[tyAlmData.udiCode].sRcyText;
		END_IF

		sStatTxt	:= tyAlmData.sAlmMsg;

	ELSIF bRstErr AND (tyAlmData.udiCode <> 0) THEN

		tyAlmData.udiCode	:= 0;
		tyAlmData.eSeverity	:= AlmSeverityNA;
		tyAlmData.sAlmMsg	:= '';
		tyAlmData.sRcyMsg	:= '';
		tyAlmData.bAlm			:= FALSE;
		sStatTxt	:= a_sStatText[eStat];

	END_IF

END_ACTION
```

#### Act_InitGlobal.st
```iecst
(** 2019-03-25 **)
ACTION Act_InitGlobal:

	(* Always Change If Project Change *)

	//Pass Data To Link
	p_bLinkStartupRun ACCESS p_StartupRun;

	//Pass Data To Internal Use
	p_udiRstErr ACCESS p_RstErrReset;
	p_sSetIPAddr ACCESS p_UISetIPAddr;
	p_sSetSubnetMask ACCESS p_UISetSubnetMask;
	p_sDevice ACCESS p_NtParamHWInfoDevice;
	p_sProgNm ACCESS p_NtParamHWInfoProgNm;
	p_bNtSettingsLoadDone ACCESS p_StartupNtSettingsLoadDone;
	p_usiNetworkMod ACCESS p_UINetworkMode;
	(* Always Change If Project Change *)

END_ACTION
```

#### Act_Initial.st
```iecst
(** 2020-09-22 **)
ACTION Act_Initial:

	//Initial
	sStatTxt	:= a_sStatText[eStat];

	fbGetIPAddr.pDevice	:= ADR(p_sDevice);
	fbGetIPAddr.pIPAddr	:= ADR(sIPAddr);
	fbGetIPAddr.Len		:= SIZEOF(sIPAddr);
	fbGetIPAddr(enable := FALSE);

	fbGetSubnetMask.pDevice		:= ADR(p_sDevice);
	fbGetSubnetMask.pSubnetMask	:= ADR(sSubnetMask);
	fbGetSubnetMask.Len			:= SIZEOF(sSubnetMask);
	fbGetSubnetMask(enable := FALSE);

	fbGetMacAddr.pDevice	:= ADR(p_sDevice);
	fbGetMacAddr.pMacAddr	:= ADR(a_usiMacAddr);
	fbGetMacAddr.Len		:= SIZEOF(a_usiMacAddr);
	fbGetMacAddr(enable := FALSE);

	fbSetIPAddr.pDevice	:= ADR(p_sDevice);
	fbSetIPAddr.pIPAddr	:= ADR(p_sSetIPAddr);
	fbSetIPAddr.Option	:= cfgOPTION_NON_VOLATILE;
	fbSetIPAddr(enable := FALSE);

	fbSetSubnetMask.pDevice		:= ADR(p_sDevice);
	fbSetSubnetMask.pSubnetMask	:= ADR(p_sSetSubnetMask);
	fbSetSubnetMask.Option		:= cfgOPTION_NON_VOLATILE;
	fbSetSubnetMask(enable := FALSE);

	fbGetETHConfigMode.pDevice	:= ADR(p_sDevice);
	fbGetETHConfigMode(enable := FALSE);

	fbSetETHConfigMode.pDevice		:= ADR(p_sDevice);
	fbSetETHConfigMode.Option		:= cfgOPTION_NON_VOLATILE;
	fbSetETHConfigMode(enable := FALSE);

END_ACTION
```

#### Act_InitLocal.st
```iecst
(** 2020-09-22 **)
ACTION Act_InitLocal:

	//Input Reference Link To Local Variable
	p_eAct ACCESS ADR(eAct);
	p_udiRstErr ACCESS ADR(udiRstErr);
	p_sSetIPAddr ACCESS ADR(sSetIPAddr);
	p_sSetSubnetMask ACCESS ADR(sSetSubnetMask);
	p_sDevice ACCESS ADR(sDevice);
	p_sProgNm ACCESS ADR(sProgNm);
	p_bNtSettingsLoadDone ACCESS ADR(bNtSettingsLoadDone);
	p_usiNetworkMod ACCESS ADR(usiNetworkMode);

END_ACTION
```

#### Act_Link.st
```iecst
(** 2019-03-29 **)
ACTION Act_Link:

END_ACTION
```

#### Act_LinkAction.st
```iecst
(** 2019-03-29 **)
ACTION Act_LinkAction:

	IF p_bLinkStartupRun = TRUE THEN
		p_eAct ACCESS p_StartupHWInfoAct;
	ELSE
		p_eAct ACCESS p_UIHWInfoAct;
	END_IF

END_ACTION
```

#### Act_Main.st
```iecst
(** 2020-10-05 **)
ACTION Act_Main:

	//Main
	CASE eStat OF

		HWInfoActIdle:
			IF eStatus <> Idle THEN	//Reset Data
				//Private
				fbGetIPAddr(enable := FALSE);
				fbGetMacAddr(enable := FALSE);
				fbSetIPAddr(enable := FALSE);
				fbSetSubnetMask(enable := FALSE);
				fbGetETHConfigMode(enable := FALSE);
				fbSetETHConfigMode(enable := FALSE);

				sStatTxt	:= a_sStatText[eStat];

			END_IF

			eStatus	:= Idle;

		HWInfoActGetIPAddr:
			IF eStatus = Idle OR eStatus = Busy THEN

				eStatus	:= Busy;

				sStatTxt	:= a_sStatText[eStat];

				IF DiagCpuIsSimulated() = FALSE THEN
					fbGetIPAddr(enable := TRUE);
					IF fbGetIPAddr.status = 0 THEN
						eStatus	:= Done;
					ELSIF fbGetIPAddr.status < 65534 THEN
						udiStatus	:= 10000;	//Get IP Address Error
						eStatus		:= Error;
					END_IF

				ELSE
					eStatus	:= Done;
					sIPAddr	:= '127.0.0.1';

				END_IF

			END_IF

		HWInfoActGetSubnetMask:
			IF eStatus = Idle OR eStatus = Busy THEN

				eStatus	:= Busy;

				sStatTxt	:= a_sStatText[eStat];

				IF DiagCpuIsSimulated() = FALSE THEN
					fbGetSubnetMask(enable := TRUE);
					IF fbGetSubnetMask.status = 0 THEN
						eStatus	:= Done;
					ELSIF fbGetSubnetMask.status < 65534 THEN
						udiStatus	:= 10001;	//Get Subnet Mask Error
						eStatus		:= Error;
					END_IF

				ELSE
					eStatus		:= Done;
					sSubnetMask	:= '255.255.0.0';

				END_IF

			END_IF

		HWInfoActGetMacAddr:
			IF eStatus = Idle OR eStatus = Busy THEN

				eStatus	:= Busy;

				sStatTxt	:= a_sStatText[eStat];

				IF DiagCpuIsSimulated() = FALSE THEN
					fbGetMacAddr(enable := TRUE);
					IF fbGetMacAddr.status = 0 THEN
						eStatus	:= Done;
					ELSIF fbGetMacAddr.status < 65534 THEN
						udiStatus	:= 10002;	//Get Mac Address Error
						eStatus		:= Error;
					END_IF

				ELSE
					eStatus	:= Done;

				END_IF

			END_IF

		HWInfoActSetIPAddr:
			IF eStatus = Idle OR eStatus = Busy THEN

				eStatus	:= Busy;

				sStatTxt	:= a_sStatText[eStat];

				IF DiagCpuIsSimulated() = FALSE THEN
					fbSetIPAddr(enable := TRUE);
					IF fbSetIPAddr.status = 0 THEN
						sIPAddr	:= p_sSetIPAddr;
						eStatus	:= Done;
					ELSIF fbSetIPAddr.status < 65534 THEN
						udiStatus	:= 10003;	//Set IP Address Error
						eStatus		:= Error;
					END_IF

				ELSE
					eStatus	:= Done;

				END_IF

			END_IF

		HWInfoActSetSubnetMask:
			IF eStatus = Idle OR eStatus = Busy THEN

				eStatus	:= Busy;

				sStatTxt	:= a_sStatText[eStat];

				IF DiagCpuIsSimulated() = FALSE THEN
					fbSetSubnetMask(enable := TRUE);
					IF fbSetSubnetMask.status = 0 THEN
						sSubnetMask	:= p_sSetSubnetMask;
						eStatus		:= Done;
					ELSIF fbSetSubnetMask.status < 65534 THEN
						udiStatus	:= 10004;	//Set Subnet Mask Error
						eStatus		:= Error;
					END_IF

				ELSE
					eStatus	:= Done;

				END_IF

			END_IF

		HWInfoActGetEthConfigMode:
			IF eStatus = Idle OR eStatus = Busy THEN

				eStatus	:= Busy;

				sStatTxt	:= a_sStatText[eStat];

				IF DiagCpuIsSimulated() = FALSE THEN
					fbGetETHConfigMode(enable := TRUE);
					IF fbGetETHConfigMode.status = 0 THEN
						udiConfigMode := fbGetETHConfigMode.ConfigMode;
						eStatus	:= Done;
					ELSIF fbGetETHConfigMode.status < 65534 THEN
						udiStatus	:= 10005;	//Get Network Configuration  Error
						eStatus		:= Error;
					END_IF

				ELSE
					eStatus	:= Done;

				END_IF

			END_IF

		HWInfoActSetEthConfigMode:
			IF eStatus = Idle OR eStatus = Busy THEN

				eStatus	:= Busy;

				sStatTxt	:= a_sStatText[eStat];

				IF DiagCpuIsSimulated() = FALSE THEN
					fbSetETHConfigMode.ConfigMode := USINT_TO_UDINT(p_usiNetworkMod);
					fbSetETHConfigMode(enable := TRUE);

					IF fbSetETHConfigMode.status = 0 THEN
						eStatus	:= Done;
					ELSIF fbSetETHConfigMode.status < 65534 THEN
						udiStatus	:= 10006;	//Set Network Configuration  Error
						eStatus		:= Error;
					END_IF

				ELSE
					eStatus	:= Done;

				END_IF

			END_IF

	END_CASE

END_ACTION
```

#### Init.st
```iecst
(** 2020-09-22 **)
PROGRAM _INIT

	(* Always Change If Project Change *)

	//Pass Address To Global Address For External Use
	//Action, State & Status
	p_HWInfoStat	:= ADR(eStat);
	p_HWInfoStatus	:= ADR(eStatus);
	p_HWInfoStatTxt	:= ADR(sStatTxt);

	//Alarm
	p_HWInfoAlmData	:= ADR(tyAlmData);

	//Output
	p_HWInfoIPAddr		:= ADR(sIPAddr);
	p_HWInfoSubnetMask	:= ADR(sSubnetMask);
	p_HWInfoMacAddr		:= ADR(a_usiMacAddr);
	p_HWInfoEthMode		:= ADR(udiConfigMode);

	(* Always Change If Project Change *)

END_PROGRAM
```

### TLBuz.typ - Do Not Change!!!
```iecst
(*2019-05-20*)
(**)
(*Action*)

TYPE
	eTLBuzAction :
		(
		TLBuzActIdle,
		TLBuzActSetGreen,
		TLBuzActSetAmber,
		TLBuzActSetRed,
		TLBuzActSetWhite,
		TLBuzActSetBlue,
		TLBuzActSetBuz,
		TLBuzActRstGreen,
		TLBuzActRstAmber,
		TLBuzActRstRed,
		TLBuzActRstWhite,
		TLBuzActRstBlue,
		TLBuzActRstBuz,
		TLBuzActSetAll,
		TLBuzActRstAll
		);
	eTLBuzMod :
		(
		TLBuzModNutek,
		TLBuzModMEK,
		TLBuzModBHTC,
		TLBuzModAptiv
		);
END_TYPE
```

### TLBuz.var - Change By Project
```iecst
(*2019-03-25*)
(**)
(*Action & State & Status*)
VAR
	p_TLBuzStat : UDINT;
	p_TLBuzStatus : UDINT;
	p_TLBuzStatTxt : UDINT;
END_VAR
(**)
(*Alarm*)
(**)
(*Output*)
VAR
	p_TLBuzRed : UDINT;
	p_TLBuzAmber : UDINT;
	p_TLBuzGreen : UDINT;
	p_TLBuzBlue : UDINT;
	p_TLBuzWhite : UDINT;
	p_TLBuzBeep : UDINT;
END_VAR
```

### Program Logical/TLBuz/TLBuz (IEC, version 1.00.0) - 1.00.0 - NtTLBuz v5.00.0

#### Init.st - Change By Project
```iecst
(** 2019-03-25 **)
PROGRAM _INIT

	(* Always Change If Project Change *)

	//Pass Address To Global Address For External Use
	//Action, State & Status
	p_TLBuzStat		:= ADR(eStat);
	p_TLBuzStatus	:= ADR(eStatus);
	p_TLBuzStatTxt	:= ADR(sStatTxt);

	//Alarm

	//Output
	p_TLBuzBlue		:= ADR(bTLBlue);
	p_TLBuzRed		:= ADR(bTLRed);
	p_TLBuzAmber	:= ADR(bTLAmber);
	p_TLBuzWhite	:= ADR(bTLWhite);
	p_TLBuzGreen	:= ADR(bTLGreen);
	p_TLBuzBeep		:= ADR(bBuzBeep);

	(* Always Change If Project Change *)

END_PROGRAM
```

#### Act_InitGlobal.st - Change By Project
```iecst
(** 2019-05-20 **)
ACTION Act_InitGlobal:

	(* Always Change If Project Change *)

	//Pass Data To Link
	p_bLinkAlarmWarning ACCESS p_AlarmWarning;
	p_bLinkAlarmInfo ACCESS p_AlarmInfo;
	p_bLinkAlarmInfoLF ACCESS p_AlarmInfoLF;
	p_bLinkLFBuzMute ACCESS p_McParamLFBuzMute;

	//Pass Data To Internal Use
	p_bManual ACCESS p_UIUIMnlMod;
	p_bStartup ACCESS p_StartupRun;
	p_bErr ACCESS p_AlarmErr;
	p_bSeqStop ACCESS p_OpsStatusCycleStop;
	p_bStep ACCESS p_OpsStatusStep;
	p_bOps ACCESS p_OpsStatusRun;
	p_bStandby ACCESS p_OpsStatusStop;
	p_bMuteBuz ACCESS p_UIMuteBuz;
	// ADD START
	p_tTLChgRcpBlinkTm ACCESS p_NtParamTLChgRcpBlinkTm;

	p_tTLErrBlinkTm ACCESS p_NtParamTLErrBlinkTm;
	p_tBuzErrOnTm ACCESS p_NtParamBuzErrOnTm;
	p_tBuzErrRestTm ACCESS p_NtParamBuzErrRestTm;
	p_usiBuzErrOnCntr ACCESS p_NtParamBuzErrOnCntr;
	p_bBuzErrStopSeqEn ACCESS p_NtParamBuzErrStopSeqEn;
	p_usiBuzErrStopSeqCntr ACCESS p_NtParamBuzErrStopSeqCntr;

	p_tTLWarnBlinkTm ACCESS p_NtParamTLWarnBlinkTm;
	p_tBuzWarnOnTm ACCESS p_NtParamBuzWarnOnTm;
	p_tBuzWarnRestTm ACCESS p_NtParamBuzWarnRestTm;
	p_usiBuzWarnOnCntr ACCESS p_NtParamBuzWarnOnCntr;
	p_bBuzWarnStopSeqEn ACCESS p_NtParamBuzWarnStopSeqEn;
	p_usiBuzWarnStopSeqCntr ACCESS p_NtParamBuzWarnStopSeqCntr;

	p_tTLWarn1BlinkTm ACCESS p_NtParamTLWarn1BlinkTm;
	p_tBuzWarn1OnTm ACCESS p_NtParamBuzWarn1OnTm;
	p_tBuzWarn1RestTm ACCESS p_NtParamBuzWarn1RestTm;
	p_usiBuzWarn1OnCntr ACCESS p_NtParamBuzWarn1OnCntr;
	p_bBuzWarn1StopSeqEn ACCESS p_NtParamBuzWarn1StopSeqEn;
	p_usiBuzWarn1StopSeqCntr ACCESS p_NtParamBuzWarn1StopSeqCntr;

	p_tTLWarn2BlinkTm ACCESS p_NtParamTLWarn2BlinkTm;
	p_tBuzWarn2OnTm ACCESS p_NtParamBuzWarn2OnTm;
	p_tBuzWarn2RestTm ACCESS p_NtParamBuzWarn2RestTm;
	p_usiBuzWarn2OnCntr ACCESS p_NtParamBuzWarn2OnCntr;
	p_bBuzWarn2StopSeqEn ACCESS p_NtParamBuzWarn2StopSeqEn;
	p_usiBuzWarn2StopSeqCntr ACCESS p_NtParamBuzWarn2StopSeqCntr;

	p_tTLWarn3BlinkTm ACCESS p_NtParamTLWarn3BlinkTm;
	p_tBuzWarn3OnTm ACCESS p_NtParamBuzWarn3OnTm;
	p_tBuzWarn3RestTm ACCESS p_NtParamBuzWarn3RestTm;
	p_usiBuzWarn3OnCntr ACCESS p_NtParamBuzWarn3OnCntr;
	p_bBuzWarn3StopSeqEn ACCESS p_NtParamBuzWarn3StopSeqEn;
	p_usiBuzWarn3StopSeqCntr ACCESS p_NtParamBuzWarn3StopSeqCntr;

	p_tTLWarn4BlinkTm ACCESS p_NtParamTLWarn4BlinkTm;
	p_tBuzWarn4OnTm ACCESS p_NtParamBuzWarn4OnTm;
	p_tBuzWarn4RestTm ACCESS p_NtParamBuzWarn4RestTm;
	p_usiBuzWarn4OnCntr ACCESS p_NtParamBuzWarn4OnCntr;
	p_bBuzWarn4StopSeqEn ACCESS p_NtParamBuzWarn4StopSeqEn;
	p_usiBuzWarn4StopSeqCntr ACCESS p_NtParamBuzWarn4StopSeqCntr;

	p_tTLWarn5BlinkTm ACCESS p_NtParamTLWarn5BlinkTm;
	p_tBuzWarn5OnTm ACCESS p_NtParamBuzWarn5OnTm;
	p_tBuzWarn5RestTm ACCESS p_NtParamBuzWarn5RestTm;
	p_usiBuzWarn5OnCntr ACCESS p_NtParamBuzWarn5OnCntr;
	p_bBuzWarn5StopSeqEn ACCESS p_NtParamBuzWarn5StopSeqEn;
	p_usiBuzWarn5StopSeqCntr ACCESS p_NtParamBuzWarn5StopSeqCntr;

	p_tBuzAlertOnTm ACCESS p_NtParamBuzAlertOnTm;
	p_tBuzAlertRestTm ACCESS p_NtParamBuzAlertRestTm;
	p_usiBuzAlertOnCntr ACCESS p_NtParamBuzAlertOnCntr;
	p_bBuzAlertStopSeqEn ACCESS p_NtParamBuzAlertStopSeqEn;
	p_usiBuzAlertStopSeqCntr ACCESS p_NtParamBuzAlertStopSeqCntr;

	p_tTLBlueBlinkTm ACCESS p_NtParamTLBlueBlinkTm;
	p_tTLAmberBlinkTm ACCESS p_NtParamTLAmberBlinkTm;
	p_tTLWhiteBlinkTm ACCESS p_NtParamTLWhiteBlinkTm;
	p_tTLRedBlinkTm ACCESS p_NtParamTLRedBlinkTm;
	p_tTLGreenBlinkTm ACCESS p_NtParamTLGreenBlinkTm;
	// ADD END
	//p_tChgRcpBlinkTm ACCESS p_NtParamTLBuzChgRcpBlinkTm;
	//p_tWarnBlinkTm ACCESS p_NtParamTLBuzWarnBlinkTm;
	//p_tWarnRestTm ACCESS p_NtParamTLBuzWarnRestTm;
	//p_usiWarnOnTm ACCESS p_NtParamTLBuzWarnOnTm;
	//p_tWarn1BlinkTm ACCESS p_NtParamTLBuzWarn1BlinkTm;
	//p_tWarn1RestTm ACCESS p_NtParamTLBuzWarn1RestTm;
	//p_usiWarn1OnTm ACCESS p_NtParamTLBuzWarn1OnTm;
	//p_tWarn2BlinkTm ACCESS p_NtParamTLBuzWarn2BlinkTm;
	//p_tWarn2RestTm ACCESS p_NtParamTLBuzWarn2RestTm;
	//p_usiWarn2OnTm ACCESS p_NtParamTLBuzWarn2OnTm;
	//p_tWarn3BlinkTm ACCESS p_NtParamTLBuzWarn3BlinkTm;
	//p_tWarn3RestTm ACCESS p_NtParamTLBuzWarn3RestTm;
	//p_usiWarn3OnTm ACCESS p_NtParamTLBuzWarn3OnTm;
	//p_tWarn4BlinkTm ACCESS p_NtParamTLBuzWarn4BlinkTm;
	//p_tWarn4RestTm ACCESS p_NtParamTLBuzWarn4RestTm;
	//p_usiWarn4OnTm ACCESS p_NtParamTLBuzWarn4OnTm;
	//p_tWarn5BlinkTm ACCESS p_NtParamTLBuzWarn5BlinkTm;
	//p_tWarn5RestTm ACCESS p_NtParamTLBuzWarn5RestTm;
	//p_usiWarn5OnTm ACCESS p_NtParamTLBuzWarn5OnTm;

	p_bCoverSwitchSig ACCESS p_DICoverSWSig;
	p_eTLBuzMode ACCESS p_NtParamTLBuzMode;

	(* Always Change If Project Change *)

END_ACTION
```

#### InputRef_Link.var - Change By Project
```iecst
(*2019-04-09*)
(**)
VAR
	p_bLinkAlarmWarning : REFERENCE TO BOOL;
	p_bLinkAlarmInfo : REFERENCE TO BOOL;
	p_bLinkAlarmInfoLF : REFERENCE TO BOOL;
	p_bLinkLFBuzMute : REFERENCE TO BOOL;
END_VAR
```

#### Act_LinkAction.st - Change By Project
```iecst
(** 2019-04-09 **)
ACTION Act_LinkAction:

	IF p_bManual = TRUE THEN
		p_eAct ACCESS p_UITLBuzAct;
	ELSE
		p_eAct ACCESS ADR(eAct);
	END_IF

END_ACTION
```

#### Act_Link.st - Change By Project
```iecst
(** 2019-03-29 **)
ACTION Act_Link:

	p_bWarning			:= p_bLinkAlarmWarning OR (p_bLinkAlarmInfo AND NOT (p_bLinkAlarmInfoLF AND p_bLinkLFBuzMute));

	p_bWarningNoBuz		:= p_bLinkAlarmInfoLF AND p_bLinkLFBuzMute;

END_ACTION
```

#### Cyclic.st - Do Not Change!!!
```iecst
(** 2020-03-16 **)
PROGRAM _CYCLIC

	IF bInitDone = FALSE THEN
		bInitDone	:= TRUE;

		Act_InitLocal;
		Act_InitGlobal;

	ELSIF bInitialDone = FALSE THEN
		bInitialDone	:= TRUE;

		Act_Initial;

	ELSE

		Act_LinkAction;
		Act_Action;
		Act_Link;
		Act_Main;

		CASE p_eTLBuzMode OF
			TLBuzModNutek:
				Act_Background;
			TLBuzModAptiv:
				Act_Background1;
			TLBuzModMEK:
				Act_Background2;
			TLBuzModBHTC:
				Act_Background3;
		END_CASE

	END_IF

END_PROGRAM
```

#### Act_InitLocal.st - Do Not Change!!!
```iecst
(** 2020-03-16 **)
ACTION Act_InitLocal:

	//Input Reference Link To Local Variable
	p_eAct ACCESS ADR(eAct);
	p_bManual ACCESS ADR(bManual);
	p_bStartup ACCESS ADR(bStartup);
	p_bErr ACCESS ADR(bErr);
	p_bErrNoBuz ACCESS ADR(bErrNoBuz);
	p_bWarning ACCESS ADR(bWarning);
	p_bWarningNoBuz ACCESS ADR(bWarningNoBuz);
	p_bWarning1 ACCESS ADR(bWarning1);
	p_bWarning1NoBuz ACCESS ADR(bWarning1NoBuz);
	p_bWarning2 ACCESS ADR(bWarning2);
	p_bWarning2NoBuz ACCESS ADR(bWarning2NoBuz);
	p_bWarning3 ACCESS ADR(bWarning3);
	p_bWarning3NoBuz ACCESS ADR(bWarning3NoBuz);
	p_bWarning4 ACCESS ADR(bWarning4);
	p_bWarning4NoBuz ACCESS ADR(bWarning4NoBuz);
	p_bWarning5 ACCESS ADR(bWarning5);
	p_bWarning5NoBuz ACCESS ADR(bWarning5NoBuz);
	p_bChgRcp ACCESS ADR(bChgRcp);
	p_bSeqStop ACCESS ADR(bSeqStop);
	p_bStep ACCESS ADR(bStep);
	p_bOps ACCESS ADR(bOps);
	p_bStandby ACCESS ADR(bStandby);
	p_bSimulation ACCESS ADR(bSimulation);
	p_bMuteBuz ACCESS ADR(bMuteBuz);

	// ADD START
	p_tTLChgRcpBlinkTm ACCESS ADR(tTLChgRcpBlinkTm);

	p_tTLErrBlinkTm ACCESS ADR(tTLErrBlinkTm);
	p_tBuzErrOnTm ACCESS ADR(tBuzErrOnTm);
	p_tBuzErrRestTm ACCESS ADR(tBuzErrRestTm);
	p_usiBuzErrOnCntr ACCESS ADR(usiBuzErrOnCntr);
	p_bBuzErrStopSeqEn ACCESS ADR(bBuzErrStopSeqEn);
	p_usiBuzErrStopSeqCntr ACCESS ADR(usiBuzErrStopSeqCntr);

	p_tTLWarnBlinkTm ACCESS ADR(tTLWarnBlinkTm);
	p_tBuzWarnOnTm ACCESS ADR(tBuzWarnOnTm);
	p_tBuzWarnRestTm ACCESS ADR(tBuzWarnRestTm);
	p_usiBuzWarnOnCntr ACCESS ADR(usiBuzWarnOnCntr);
	p_bBuzWarnStopSeqEn ACCESS ADR(bBuzWarnStopSeqEn);
	p_usiBuzWarnStopSeqCntr ACCESS ADR(usiBuzWarnStopSeqCntr);

	p_tTLWarn1BlinkTm ACCESS ADR(tTLWarn1BlinkTm);
	p_tBuzWarn1OnTm ACCESS ADR(tBuzWarn1OnTm);
	p_tBuzWarn1RestTm ACCESS ADR(tBuzWarn1RestTm);
	p_usiBuzWarn1OnCntr ACCESS ADR(usiBuzWarn1OnCntr);
	p_bBuzWarn1StopSeqEn ACCESS ADR(bBuzWarn1StopSeqEn);
	p_usiBuzWarn1StopSeqCntr ACCESS ADR(usiBuzWarn1StopSeqCntr);

	p_tTLWarn2BlinkTm ACCESS ADR(tTLWarn2BlinkTm);
	p_tBuzWarn2OnTm ACCESS ADR(tBuzWarn2OnTm);
	p_tBuzWarn2RestTm ACCESS ADR(tBuzWarn2RestTm);
	p_usiBuzWarn2OnCntr ACCESS ADR(usiBuzWarn2OnCntr);
	p_bBuzWarn2StopSeqEn ACCESS ADR(bBuzWarn2StopSeqEn);
	p_usiBuzWarn2StopSeqCntr ACCESS ADR(usiBuzWarn2StopSeqCntr);

	p_tTLWarn3BlinkTm ACCESS ADR(tTLWarn3BlinkTm);
	p_tBuzWarn3OnTm ACCESS ADR(tBuzWarn3OnTm);
	p_tBuzWarn3RestTm ACCESS ADR(tBuzWarn3RestTm);
	p_usiBuzWarn3OnCntr ACCESS ADR(usiBuzWarn3OnCntr);
	p_bBuzWarn3StopSeqEn ACCESS ADR(bBuzWarn3StopSeqEn);
	p_usiBuzWarn3StopSeqCntr ACCESS ADR(usiBuzWarn3StopSeqCntr);

	p_tTLWarn4BlinkTm ACCESS ADR(tTLWarn4BlinkTm);
	p_tBuzWarn4OnTm ACCESS ADR(tBuzWarn4OnTm);
	p_tBuzWarn4RestTm ACCESS ADR(tBuzWarn4RestTm);
	p_usiBuzWarnOnCntr ACCESS ADR(usiBuzWarn4OnCntr);
	p_bBuzWarn4StopSeqEn ACCESS ADR(bBuzWarn4StopSeqEn);
	p_usiBuzWarn4StopSeqCntr ACCESS ADR(usiBuzWarn4StopSeqCntr);

	p_tTLWarn5BlinkTm ACCESS ADR(tTLWarn5BlinkTm);
	p_tBuzWarn5OnTm ACCESS ADR(tBuzWarn5OnTm);
	p_tBuzWarn5RestTm ACCESS ADR(tBuzWarn5RestTm);
	p_usiBuzWarn5OnCntr ACCESS ADR(usiBuzWarn5OnCntr);
	p_bBuzWarn5StopSeqEn ACCESS ADR(bBuzWarn5StopSeqEn);
	p_usiBuzWarn5StopSeqCntr ACCESS ADR(usiBuzWarn5StopSeqCntr);

	p_tBuzAlertOnTm ACCESS ADR(tBuzAlertOnTm);
	p_tBuzAlertRestTm ACCESS ADR(tBuzAlertRestTm);
	p_usiBuzAlertOnCntr ACCESS ADR(usiBuzAlertOnCntr);
	p_bBuzAlertStopSeqEn ACCESS ADR(bBuzAlertStopSeqEn);
	p_usiBuzAlertStopSeqCntr ACCESS ADR(usiBuzAlertStopSeqCntr);

	p_tTLBlueBlinkTm ACCESS ADR(tTLBlueBlinkTm);
	p_tTLAmberBlinkTm ACCESS ADR(tTLAmberBlinkTm);
	p_tTLWhiteBlinkTm ACCESS ADR(tTLWhiteBlinkTm);
	p_tTLRedBlinkTm ACCESS ADR(tTLRedBlinkTm);
	p_tTLGreenBlinkTm ACCESS ADR(tTLGreenBlinkTm);
	// ADD END

	p_tErrBlinkTm ACCESS ADR(tErrBlinkTm);
	p_tChgRcpBlinkTm ACCESS ADR(tChgRcpBlinkTm);
	p_tWarnBlinkTm ACCESS ADR(tWarnBlinkTm);
	p_tWarnRestTm ACCESS ADR(tWarnRestTm);
	p_usiWarnOnTm ACCESS ADR(usiWarnOnTm);
	p_tWarn1BlinkTm ACCESS ADR(tWarn1BlinkTm);
	p_tWarn1RestTm ACCESS ADR(tWarn1RestTm);
	p_usiWarn1OnTm ACCESS ADR(usiWarn1OnTm);
	p_tWarn2BlinkTm ACCESS ADR(tWarn2BlinkTm);
	p_tWarn2RestTm ACCESS ADR(tWarn2RestTm);
	p_usiWarn2OnTm ACCESS ADR(usiWarn2OnTm);
	p_tWarn3BlinkTm ACCESS ADR(tWarn3BlinkTm);
	p_tWarn3RestTm ACCESS ADR(tWarn3RestTm);
	p_usiWarn3OnTm ACCESS ADR(usiWarn3OnTm);
	p_tWarn4BlinkTm ACCESS ADR(tWarn4BlinkTm);
	p_tWarn4RestTm ACCESS ADR(tWarn4RestTm);
	p_usiWarn4OnTm ACCESS ADR(usiWarn4OnTm);
	p_tWarn5BlinkTm ACCESS ADR(tWarn5BlinkTm);
	p_tWarn5RestTm ACCESS ADR(tWarn5RestTm);
	p_usiWarn5OnTm ACCESS ADR(usiWarn5OnTm);

	p_bCoverSwitchSig ACCESS ADR(bCoveSwitchSig);
	p_eTLBuzMode ACCESS ADR(eTLBuzMode);

	p_bAOIErrSig ACCESS ADR(bAOIErrSig);
	p_bAOIOriginSig ACCESS ADR(bAOIOriginSig);

	p_bBuzAlertEn ACCESS ADR(bBuzAlertEn);
	p_bTLBlueFlashEn ACCESS ADR(bTLBlueFlashEn);
	p_bTLAmberFlashEn ACCESS ADR(bTLAmberFlashEn);
	p_bTLWhiteFlashEn ACCESS ADR(bTLWhiteFlashEn);
	p_bTLRedFlashEn ACCESS ADR(bTLRedFlashEn);
	p_bTLGreenFlashEn ACCESS ADR(bTLGreenFlashEn);

END_ACTION
```

#### Act_Initial.st - Do Not Change!!!
```iecst
(** 2019-03-22 **)
ACTION Act_Initial:

	//Initial
	sStatTxt	:= a_sStatText[eStat];

	fbBlink(bEn := FALSE);
	fbWarning(bEn := FALSE);

END_ACTION
```

#### Act_Action.st - Do Not Change!!!
```iecst
(** 2019-03-25 **)
ACTION Act_Action:

	//Set p_eAct
	IF eStatus = Idle OR eStatus = Busy OR eStatus = Done THEN
		eStat	:= p_eAct;
	END_IF

END_ACTION
```

#### Act_Main.st - Do Not Change!!!
```iecst
(** 2020-02-18 **)
ACTION Act_Main:

	IF eStatOld <> eStat THEN
		IF eStatOld <> TLBuzActIdle
			AND eStatOld <> TLBuzActSetGreen
			AND eStatOld <> TLBuzActSetAmber
			AND eStatOld <> TLBuzActSetRed
			AND eStatOld <> TLBuzActSetBlue
			AND eStatOld <> TLBuzActSetWhite
			AND eStatOld <> TLBuzActSetBuz
			AND eStatOld <> TLBuzActRstGreen
			AND eStatOld <> TLBuzActRstAmber
			AND eStatOld <> TLBuzActRstRed
			AND eStatOld <> TLBuzActRstBlue
			AND eStatOld <> TLBuzActRstWhite
			AND eStatOld <> TLBuzActRstBuz
			AND eStatOld <> TLBuzActSetAll
			AND eStatOld <> TLBuzActRstAll THEN

			bTLGreen	:= FALSE;
			bTLAmber	:= FALSE;
			bTLWhite	:= FALSE;
			bTLBlue		:= FALSE;
			bTLRed		:= FALSE;
			bBuzBeep	:= FALSE;

		END_IF

		sStatTxt	:= a_sStatText[eStat];

		eStatOld	:= eStat;

		eStatus		:= Busy;
	END_IF

	//Main
	CASE eStat OF

		TLBuzActIdle:
			IF eStatus <> Idle THEN	//Reset Data
				//Private

				sStatTxt	:= a_sStatText[eStat];

			END_IF

			eStatus	:= Idle;

		TLBuzActSetGreen:
			IF eStatus = Idle OR eStatus = Busy THEN

				sStatTxt	:= a_sStatText[eStat];

				bTLGreen	:= TRUE;
				eStatus		:= Done;

			END_IF

		TLBuzActSetAmber:
			IF eStatus = Idle OR eStatus = Busy THEN

				sStatTxt	:= a_sStatText[eStat];

				bTLAmber	:= TRUE;
				eStatus		:= Done;

			END_IF

		TLBuzActSetRed:
			IF eStatus = Idle OR eStatus = Busy THEN

				sStatTxt	:= a_sStatText[eStat];

				bTLRed	:= TRUE;
				eStatus	:= Done;

			END_IF

		TLBuzActSetBlue:
			IF eStatus = Idle OR eStatus = Busy THEN

				sStatTxt	:= a_sStatText[eStat];

				bTLBlue		:= TRUE;
				eStatus		:= Done;

			END_IF

		TLBuzActSetWhite:
			IF eStatus = Idle OR eStatus = Busy THEN

				sStatTxt	:= a_sStatText[eStat];

				bTLWhite	:= TRUE;
				eStatus		:= Done;

			END_IF

		TLBuzActSetBuz:
			IF eStatus = Idle OR eStatus = Busy THEN

				sStatTxt	:= a_sStatText[eStat];

				bBuzBeep	:= TRUE;
				eStatus		:= Done;

			END_IF

		TLBuzActRstGreen:
			IF eStatus = Idle OR eStatus = Busy THEN

				sStatTxt	:= a_sStatText[eStat];

				bTLGreen	:= FALSE;
				eStatus		:= Done;

			END_IF

		TLBuzActRstAmber:
			IF eStatus = Idle OR eStatus = Busy THEN

				sStatTxt	:= a_sStatText[eStat];

				bTLAmber	:= FALSE;
				eStatus		:= Done;

			END_IF

		TLBuzActRstRed:
			IF eStatus = Idle OR eStatus = Busy THEN

				sStatTxt	:= a_sStatText[eStat];

				bTLRed		:= FALSE;
				eStatus		:= Done;

			END_IF

		TLBuzActRstBlue:
			IF eStatus = Idle OR eStatus = Busy THEN

				sStatTxt	:= a_sStatText[eStat];

				bTLBlue		:= FALSE;
				eStatus		:= Done;

			END_IF

		TLBuzActRstWhite:
			IF eStatus = Idle OR eStatus = Busy THEN

				sStatTxt	:= a_sStatText[eStat];

				bTLWhite	:= FALSE;
				eStatus		:= Done;

			END_IF

		TLBuzActRstBuz:
			IF eStatus = Idle OR eStatus = Busy THEN

				sStatTxt	:= a_sStatText[eStat];

				bBuzBeep	:= FALSE;
				eStatus		:= Done;

			END_IF

		TLBuzActSetAll:
			IF eStatus = Idle OR eStatus = Busy THEN

				sStatTxt	:= a_sStatText[eStat];

				bTLGreen	:= TRUE;
				bTLRed		:= TRUE;
				bTLAmber	:= TRUE;
				bTLWhite	:= TRUE;
				bTLBlue		:= TRUE;
				bBuzBeep	:= TRUE;
				eStatus		:= Done;

			END_IF

		TLBuzActRstAll:
			IF eStatus = Idle OR eStatus = Busy THEN

				sStatTxt	:= a_sStatText[eStat];

				bTLGreen	:= FALSE;
				bTLAmber	:= FALSE;
				bTLRed		:= FALSE;
				bTLWhite	:= FALSE;
				bTLBlue		:= FALSE;
				bBuzBeep	:= FALSE;
				eStatus		:= Done;

			END_IF

	END_CASE

END_ACTION
```
